// Mitsubishi GX Developer project: PLC_PCO520L2   PLC: Q06UDEH

PROGRAM OUTPUT
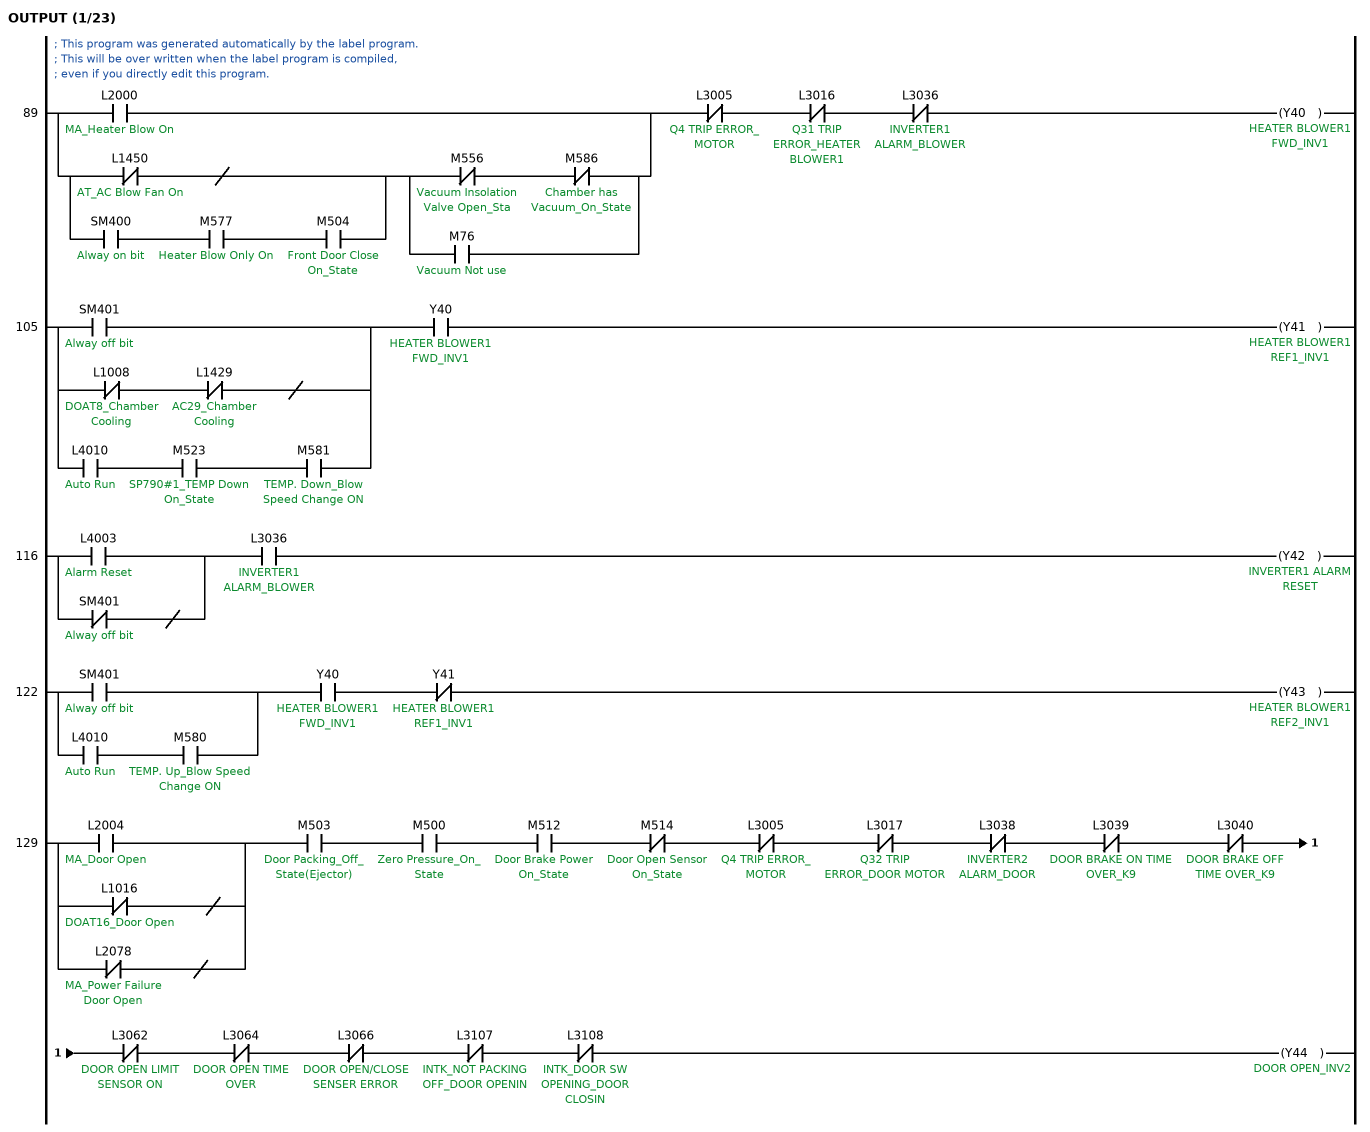
; This program was generated automatically by the label program.
; This will be over written when the label program is compiled,
; even if you directly edit this program.
89    LD      L2000  ; MA_Heater Blow On
      LDI     L1450  ; AT_AC Blow Fan On
      INV
      LD      SM400  ; Alway on bit
      AND     M577  ; Heater Blow Only On
      AND     M504  ; Front Door Close On_State
      ORB
      LDI     M556  ; Vacuum Insolation Valve Open_Sta
      ANI     M586  ; Chamber has Vacuum_On_State
      OR      M76  ; Vacuum Not use
      ANB
      ORB
      ANI     L3005  ; Q4 TRIP ERROR_MOTOR
      ANI     L3016  ; Q31 TRIP ERROR_HEATER BLOWER1
      ANI     L3036  ; INVERTER1 ALARM_BLOWER
      OUT     Y40  ; HEATER BLOWER1 FWD_INV1
105   LD      SM401  ; Alway off bit
      LDI     L1008  ; DOAT8_Chamber Cooling
      ANI     L1429  ; AC29_Chamber Cooling
      INV
      ORB
      LD      L4010  ; Auto Run
      AND     M523  ; SP790#1_TEMP Down On_State
      AND     M581  ; TEMP. Down_Blow Speed Change ON
      ORB
      AND     Y40  ; HEATER BLOWER1 FWD_INV1
      OUT     Y41  ; HEATER BLOWER1 REF1_INV1
116   LD      L4003  ; Alarm Reset
      LDI     SM401  ; Alway off bit
      INV
      ORB
      AND     L3036  ; INVERTER1 ALARM_BLOWER
      OUT     Y42  ; INVERTER1 ALARM RESET
122   LD      SM401  ; Alway off bit
      LD      L4010  ; Auto Run
      AND     M580  ; TEMP. Up_Blow Speed Change ON
      ORB
      AND     Y40  ; HEATER BLOWER1 FWD_INV1
      ANI     Y41  ; HEATER BLOWER1 REF1_INV1
      OUT     Y43  ; HEATER BLOWER1 REF2_INV1
129   LD      L2004  ; MA_Door Open
      LDI     L1016  ; DOAT16_Door Open
      INV
      ORB
      LDI     L2078  ; MA_Power Failure Door Open
      INV
      ORB
      AND     M503  ; Door Packing_Off_State(Ejector)
      AND     M500  ; Zero Pressure_On_State
      AND     M512  ; Door Brake Power On_State
      ANI     M514  ; Door Open Sensor On_State
      ANI     L3005  ; Q4 TRIP ERROR_MOTOR
      ANI     L3017  ; Q32 TRIP ERROR_DOOR MOTOR
      ANI     L3038  ; INVERTER2 ALARM_DOOR
      ANI     L3039  ; DOOR BRAKE ON TIME OVER_K9
      ANI     L3040  ; DOOR BRAKE OFF TIME OVER_K9
      ANI     L3062  ; DOOR OPEN LIMIT SENSOR ON
      ANI     L3064  ; DOOR OPEN TIME OVER
      ANI     L3066  ; DOOR OPEN/CLOSE SENSER ERROR
      ANI     L3107  ; INTK_NOT PACKING OFF_DOOR OPENIN
      ANI     L3108  ; INTK_DOOR SW OPENING_DOOR CLOSIN
      OUT     Y44  ; DOOR OPEN_INV2
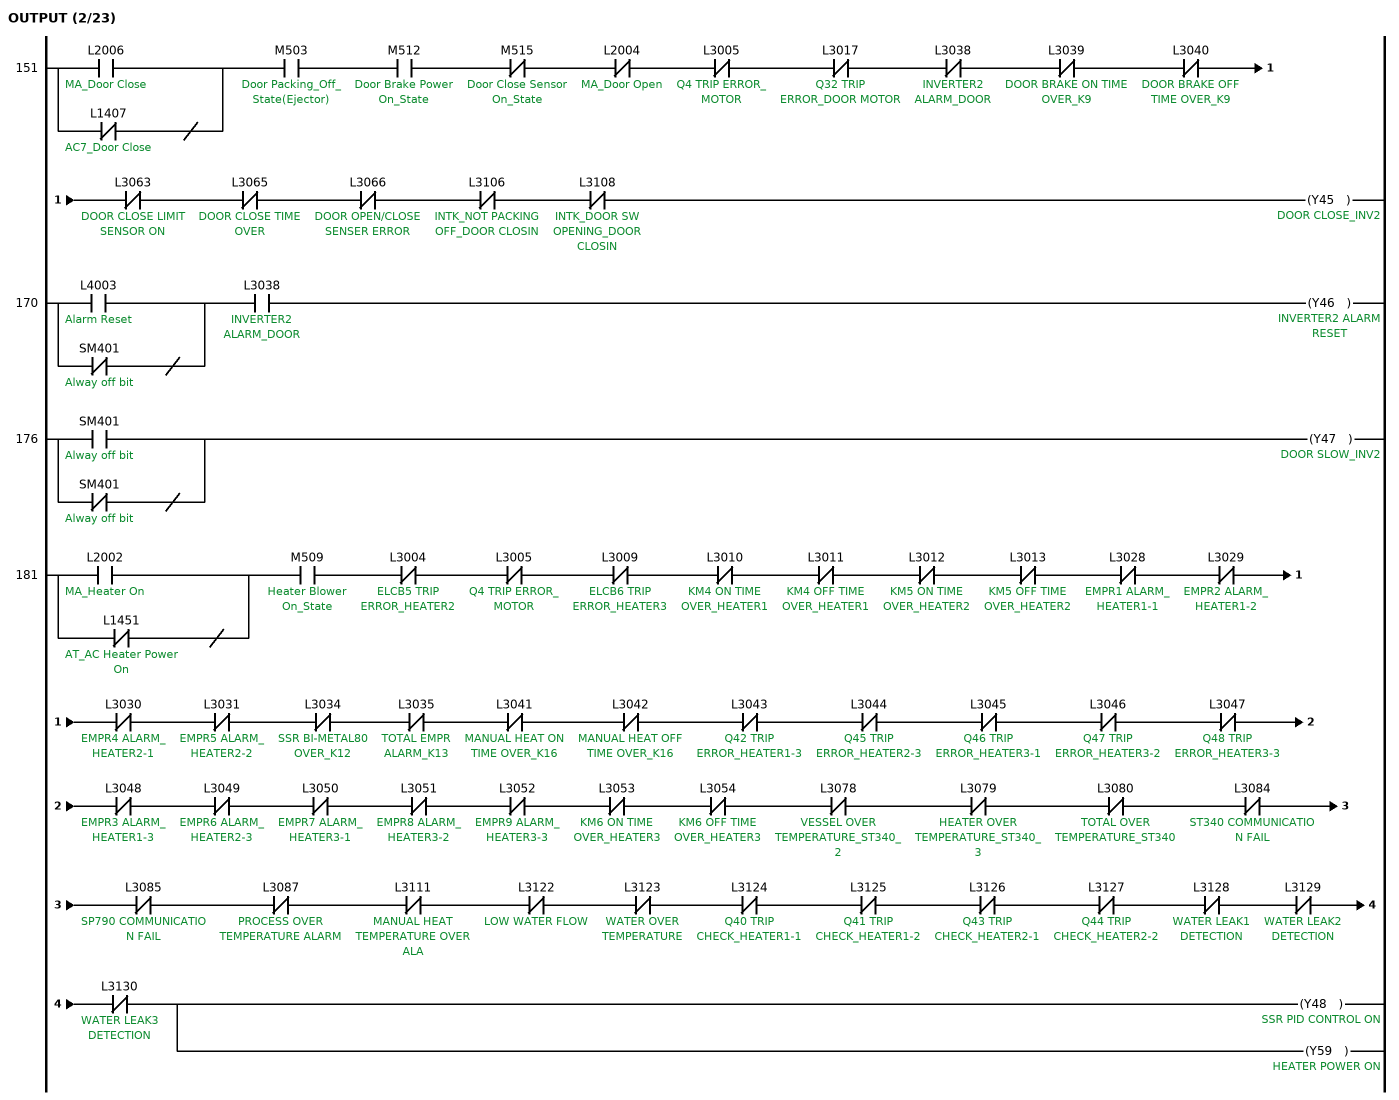
151   LD      L2006  ; MA_Door Close
      LDI     L1407  ; AC7_Door Close
      INV
      ORB
      AND     M503  ; Door Packing_Off_State(Ejector)
      AND     M512  ; Door Brake Power On_State
      ANI     M515  ; Door Close Sensor On_State
      ANI     L2004  ; MA_Door Open
      ANI     L3005  ; Q4 TRIP ERROR_MOTOR
      ANI     L3017  ; Q32 TRIP ERROR_DOOR MOTOR
      ANI     L3038  ; INVERTER2 ALARM_DOOR
      ANI     L3039  ; DOOR BRAKE ON TIME OVER_K9
      ANI     L3040  ; DOOR BRAKE OFF TIME OVER_K9
      ANI     L3063  ; DOOR CLOSE LIMIT SENSOR ON
      ANI     L3065  ; DOOR CLOSE TIME OVER
      ANI     L3066  ; DOOR OPEN/CLOSE SENSER ERROR
      ANI     L3106  ; INTK_NOT PACKING OFF_DOOR CLOSIN
      ANI     L3108  ; INTK_DOOR SW OPENING_DOOR CLOSIN
      OUT     Y45  ; DOOR CLOSE_INV2
170   LD      L4003  ; Alarm Reset
      LDI     SM401  ; Alway off bit
      INV
      ORB
      AND     L3038  ; INVERTER2 ALARM_DOOR
      OUT     Y46  ; INVERTER2 ALARM RESET
176   LD      SM401  ; Alway off bit
      LDI     SM401  ; Alway off bit
      INV
      ORB
      OUT     Y47  ; DOOR SLOW_INV2
181   LD      L2002  ; MA_Heater On
      LDI     L1451  ; AT_AC Heater Power On
      INV
      ORB
      AND     M509  ; Heater Blower On_State
      ANI     L3004  ; ELCB5 TRIP ERROR_HEATER2
      ANI     L3005  ; Q4 TRIP ERROR_MOTOR
      ANI     L3009  ; ELCB6 TRIP ERROR_HEATER3
      ANI     L3010  ; KM4 ON TIME OVER_HEATER1
      ANI     L3011  ; KM4 OFF TIME OVER_HEATER1
      ANI     L3012  ; KM5 ON TIME OVER_HEATER2
      ANI     L3013  ; KM5 OFF TIME OVER_HEATER2
      ANI     L3028  ; EMPR1 ALARM_HEATER1-1
      ANI     L3029  ; EMPR2 ALARM_HEATER1-2
      ANI     L3030  ; EMPR4 ALARM_HEATER2-1
      ANI     L3031  ; EMPR5 ALARM_HEATER2-2
      ANI     L3034  ; SSR BI-METAL80 OVER_K12
      ANI     L3035  ; TOTAL EMPR ALARM_K13
      ANI     L3041  ; MANUAL HEAT ON TIME OVER_K16
      ANI     L3042  ; MANUAL HEAT OFF TIME OVER_K16
      ANI     L3043  ; Q42 TRIP ERROR_HEATER1-3
      ANI     L3044  ; Q45 TRIP ERROR_HEATER2-3
      ANI     L3045  ; Q46 TRIP ERROR_HEATER3-1
      ANI     L3046  ; Q47 TRIP ERROR_HEATER3-2
      ANI     L3047  ; Q48 TRIP ERROR_HEATER3-3
      ANI     L3048  ; EMPR3 ALARM_HEATER1-3
      ANI     L3049  ; EMPR6 ALARM_HEATER2-3
      ANI     L3050  ; EMPR7 ALARM_HEATER3-1
      ANI     L3051  ; EMPR8 ALARM_HEATER3-2
      ANI     L3052  ; EMPR9 ALARM_HEATER3-3
      ANI     L3053  ; KM6 ON TIME OVER_HEATER3
      ANI     L3054  ; KM6 OFF TIME OVER_HEATER3
      ANI     L3078  ; VESSEL OVER TEMPERATURE_ST340_2
      ANI     L3079  ; HEATER OVER TEMPERATURE_ST340_3
      ANI     L3080  ; TOTAL OVER TEMPERATURE_ST340
      ANI     L3084  ; ST340 COMMUNICATION FAIL
      ANI     L3085  ; SP790 COMMUNICATION FAIL
      ANI     L3087  ; PROCESS OVER TEMPERATURE ALARM
      ANI     L3111  ; MANUAL HEAT TEMPERATURE OVER ALA
      ANI     L3122  ; LOW WATER FLOW
      ANI     L3123  ; WATER OVER TEMPERATURE
      ANI     L3124  ; Q40 TRIP CHECK_HEATER1-1
      ANI     L3125  ; Q41 TRIP CHECK_HEATER1-2
      ANI     L3126  ; Q43 TRIP CHECK_HEATER2-1
      ANI     L3127  ; Q44 TRIP CHECK_HEATER2-2
      ANI     L3128  ; WATER LEAK1 DETECTION
      ANI     L3129  ; WATER LEAK2 DETECTION
      ANI     L3130  ; WATER LEAK3 DETECTION
      OUT     Y48  ; SSR PID CONTROL ON
      OUT     Y59  ; HEATER POWER ON
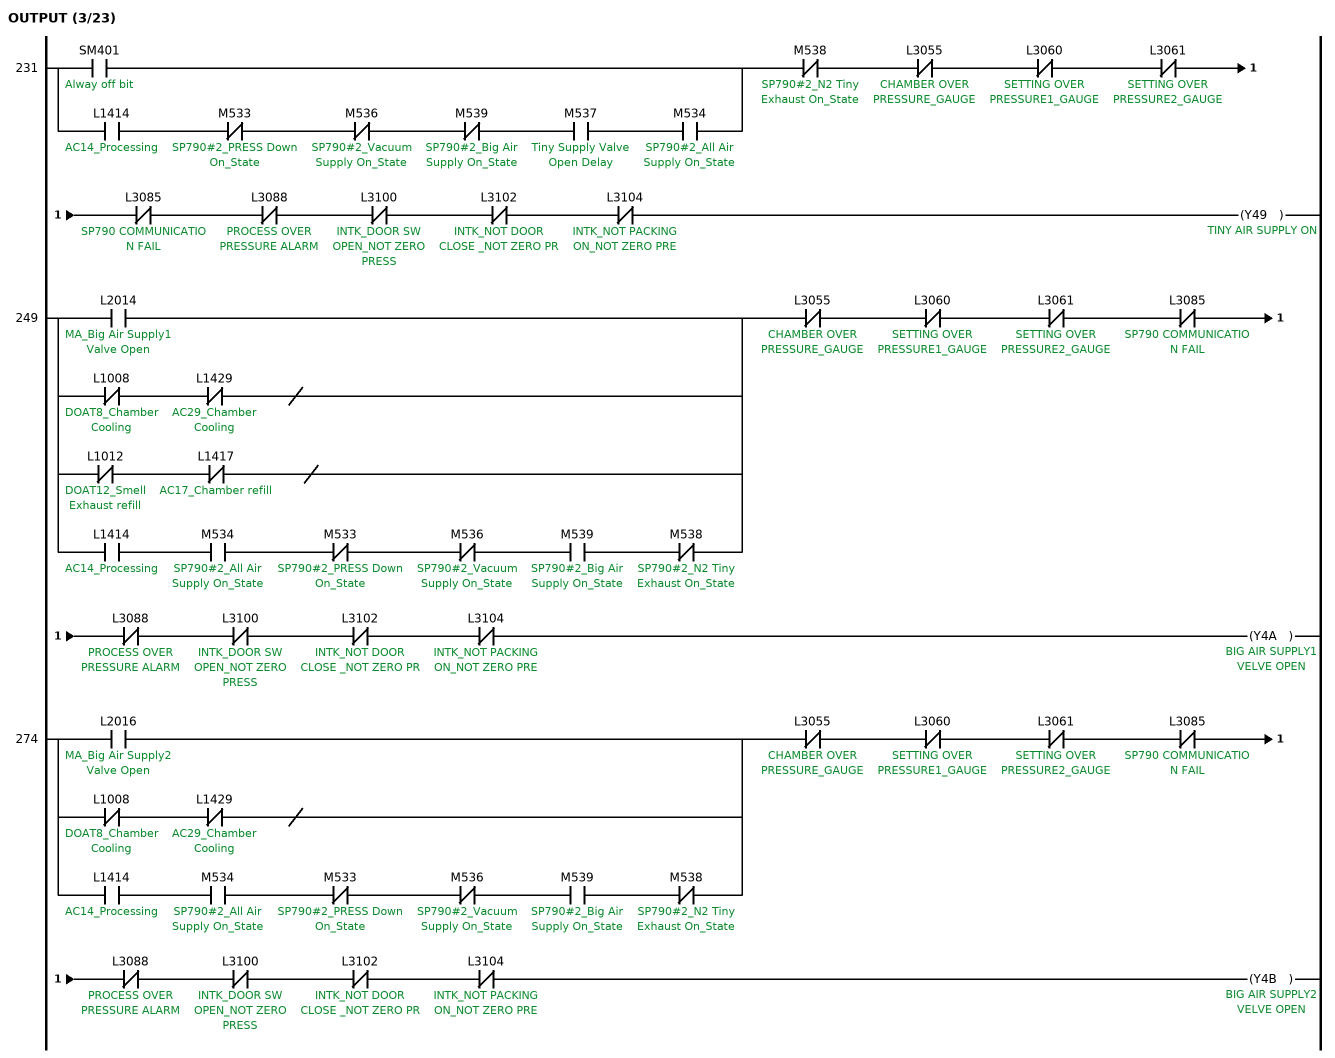
231   LD      SM401  ; Alway off bit
      LD      L1414  ; AC14_Processing
      ANI     M533  ; SP790#2_PRESS Down On_State
      ANI     M536  ; SP790#2_Vacuum Supply On_State
      ANI     M539  ; SP790#2_Big Air Supply On_State
      AND     M537  ; Tiny Supply Valve Open Delay
      AND     M534  ; SP790#2_All Air Supply On_State
      ORB
      ANI     M538  ; SP790#2_N2 Tiny Exhaust On_State
      ANI     L3055  ; CHAMBER OVER PRESSURE_GAUGE
      ANI     L3060  ; SETTING OVER PRESSURE1_GAUGE
      ANI     L3061  ; SETTING OVER PRESSURE2_GAUGE
      ANI     L3085  ; SP790 COMMUNICATION FAIL
      ANI     L3088  ; PROCESS OVER PRESSURE ALARM
      ANI     L3100  ; INTK_DOOR SW OPEN_NOT ZERO PRESS
      ANI     L3102  ; INTK_NOT DOOR CLOSE _NOT ZERO PR
      ANI     L3104  ; INTK_NOT PACKING ON_NOT ZERO PRE
      OUT     Y49  ; TINY AIR SUPPLY ON
249   LD      L2014  ; MA_Big Air Supply1 Valve Open
      LDI     L1008  ; DOAT8_Chamber Cooling
      ANI     L1429  ; AC29_Chamber Cooling
      INV
      ORB
      LDI     L1012  ; DOAT12_Smell Exhaust refill
      ANI     L1417  ; AC17_Chamber refill
      INV
      ORB
      LD      L1414  ; AC14_Processing
      AND     M534  ; SP790#2_All Air Supply On_State
      ANI     M533  ; SP790#2_PRESS Down On_State
      ANI     M536  ; SP790#2_Vacuum Supply On_State
      AND     M539  ; SP790#2_Big Air Supply On_State
      ANI     M538  ; SP790#2_N2 Tiny Exhaust On_State
      ORB
      ANI     L3055  ; CHAMBER OVER PRESSURE_GAUGE
      ANI     L3060  ; SETTING OVER PRESSURE1_GAUGE
      ANI     L3061  ; SETTING OVER PRESSURE2_GAUGE
      ANI     L3085  ; SP790 COMMUNICATION FAIL
      ANI     L3088  ; PROCESS OVER PRESSURE ALARM
      ANI     L3100  ; INTK_DOOR SW OPEN_NOT ZERO PRESS
      ANI     L3102  ; INTK_NOT DOOR CLOSE _NOT ZERO PR
      ANI     L3104  ; INTK_NOT PACKING ON_NOT ZERO PRE
      OUT     Y4A  ; BIG AIR SUPPLY1 VELVE OPEN
274   LD      L2016  ; MA_Big Air Supply2 Valve Open
      LDI     L1008  ; DOAT8_Chamber Cooling
      ANI     L1429  ; AC29_Chamber Cooling
      INV
      ORB
      LD      L1414  ; AC14_Processing
      AND     M534  ; SP790#2_All Air Supply On_State
      ANI     M533  ; SP790#2_PRESS Down On_State
      ANI     M536  ; SP790#2_Vacuum Supply On_State
      AND     M539  ; SP790#2_Big Air Supply On_State
      ANI     M538  ; SP790#2_N2 Tiny Exhaust On_State
      ORB
      ANI     L3055  ; CHAMBER OVER PRESSURE_GAUGE
      ANI     L3060  ; SETTING OVER PRESSURE1_GAUGE
      ANI     L3061  ; SETTING OVER PRESSURE2_GAUGE
      ANI     L3085  ; SP790 COMMUNICATION FAIL
      ANI     L3088  ; PROCESS OVER PRESSURE ALARM
      ANI     L3100  ; INTK_DOOR SW OPEN_NOT ZERO PRESS
      ANI     L3102  ; INTK_NOT DOOR CLOSE _NOT ZERO PR
      ANI     L3104  ; INTK_NOT PACKING ON_NOT ZERO PRE
      OUT     Y4B  ; BIG AIR SUPPLY2 VELVE OPEN
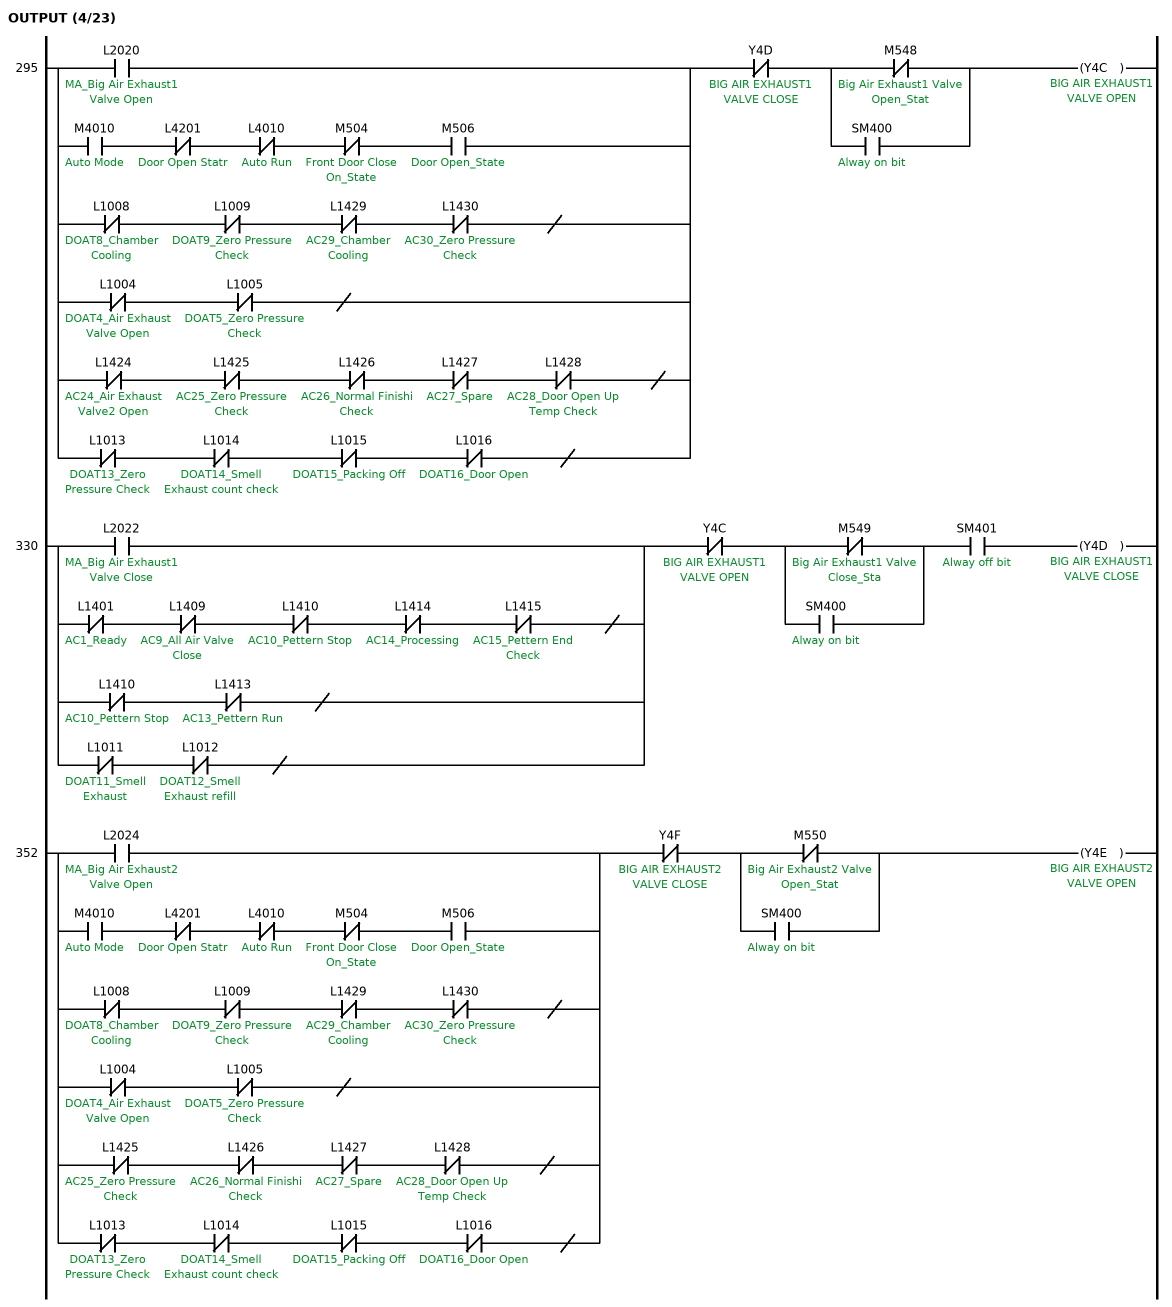
295   LD      L2020  ; MA_Big Air Exhaust1 Valve Open
      LD      M4010  ; Auto Mode
      ANI     L4201  ; Door Open Statr
      ANI     L4010  ; Auto Run
      ANI     M504  ; Front Door Close On_State
      AND     M506  ; Door Open_State
      ORB
      LDI     L1008  ; DOAT8_Chamber Cooling
      ANI     L1009  ; DOAT9_Zero Pressure Check
      ANI     L1429  ; AC29_Chamber Cooling
      ANI     L1430  ; AC30_Zero Pressure Check
      INV
      ORB
      LDI     L1004  ; DOAT4_Air Exhaust Valve Open
      ANI     L1005  ; DOAT5_Zero Pressure Check
      INV
      ORB
      LDI     L1424  ; AC24_Air Exhaust Valve2 Open
      ANI     L1425  ; AC25_Zero Pressure Check
      ANI     L1426  ; AC26_Normal Finishi Check
      ANI     L1427  ; AC27_Spare
      ANI     L1428  ; AC28_Door Open Up Temp Check
      INV
      ORB
      LDI     L1013  ; DOAT13_Zero Pressure Check
      ANI     L1014  ; DOAT14_Smell Exhaust count check
      ANI     L1015  ; DOAT15_Packing Off
      ANI     L1016  ; DOAT16_Door Open
      INV
      ORB
      ANI     Y4D  ; BIG AIR EXHAUST1 VALVE CLOSE
      LDI     M548  ; Big Air Exhaust1 Valve Open_Stat
      OR      SM400  ; Alway on bit
      ANB
      OUT     Y4C  ; BIG AIR EXHAUST1 VALVE OPEN
330   LD      L2022  ; MA_Big Air Exhaust1 Valve Close
      LDI     L1401  ; AC1_Ready
      ANI     L1409  ; AC9_All Air Valve Close
      ANI     L1410  ; AC10_Pettern Stop
      ANI     L1414  ; AC14_Processing
      ANI     L1415  ; AC15_Pettern End Check
      INV
      ORB
      LDI     L1410  ; AC10_Pettern Stop
      ANI     L1413  ; AC13_Pettern Run
      INV
      ORB
      LDI     L1011  ; DOAT11_Smell Exhaust
      ANI     L1012  ; DOAT12_Smell Exhaust refill
      INV
      ORB
      ANI     Y4C  ; BIG AIR EXHAUST1 VALVE OPEN
      LDI     M549  ; Big Air Exhaust1 Valve Close_Sta
      OR      SM400  ; Alway on bit
      ANB
      AND     SM401  ; Alway off bit
      OUT     Y4D  ; BIG AIR EXHAUST1 VALVE CLOSE
352   LD      L2024  ; MA_Big Air Exhaust2 Valve Open
      LD      M4010  ; Auto Mode
      ANI     L4201  ; Door Open Statr
      ANI     L4010  ; Auto Run
      ANI     M504  ; Front Door Close On_State
      AND     M506  ; Door Open_State
      ORB
      LDI     L1008  ; DOAT8_Chamber Cooling
      ANI     L1009  ; DOAT9_Zero Pressure Check
      ANI     L1429  ; AC29_Chamber Cooling
      ANI     L1430  ; AC30_Zero Pressure Check
      INV
      ORB
      LDI     L1004  ; DOAT4_Air Exhaust Valve Open
      ANI     L1005  ; DOAT5_Zero Pressure Check
      INV
      ORB
      LDI     L1425  ; AC25_Zero Pressure Check
      ANI     L1426  ; AC26_Normal Finishi Check
      ANI     L1427  ; AC27_Spare
      ANI     L1428  ; AC28_Door Open Up Temp Check
      INV
      ORB
      LDI     L1013  ; DOAT13_Zero Pressure Check
      ANI     L1014  ; DOAT14_Smell Exhaust count check
      ANI     L1015  ; DOAT15_Packing Off
      ANI     L1016  ; DOAT16_Door Open
      INV
      ORB
      ANI     Y4F  ; BIG AIR EXHAUST2 VALVE CLOSE
      LDI     M550  ; Big Air Exhaust2 Valve Open_Stat
      OR      SM400  ; Alway on bit
      ANB
      OUT     Y4E  ; BIG AIR EXHAUST2 VALVE OPEN
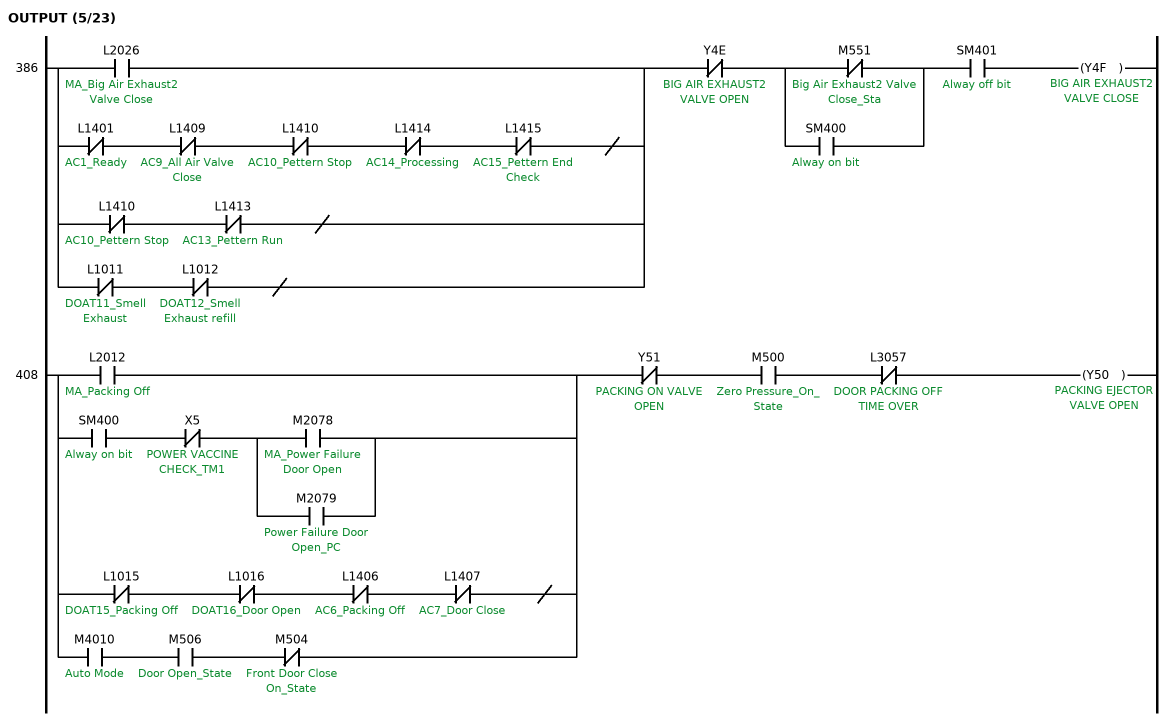
386   LD      L2026  ; MA_Big Air Exhaust2 Valve Close
      LDI     L1401  ; AC1_Ready
      ANI     L1409  ; AC9_All Air Valve Close
      ANI     L1410  ; AC10_Pettern Stop
      ANI     L1414  ; AC14_Processing
      ANI     L1415  ; AC15_Pettern End Check
      INV
      ORB
      LDI     L1410  ; AC10_Pettern Stop
      ANI     L1413  ; AC13_Pettern Run
      INV
      ORB
      LDI     L1011  ; DOAT11_Smell Exhaust
      ANI     L1012  ; DOAT12_Smell Exhaust refill
      INV
      ORB
      ANI     Y4E  ; BIG AIR EXHAUST2 VALVE OPEN
      LDI     M551  ; Big Air Exhaust2 Valve Close_Sta
      OR      SM400  ; Alway on bit
      ANB
      AND     SM401  ; Alway off bit
      OUT     Y4F  ; BIG AIR EXHAUST2 VALVE CLOSE
408   LD      L2012  ; MA_Packing Off
      LD      SM400  ; Alway on bit
      ANI     X5  ; POWER VACCINE CHECK_TM1
      LD      M2078  ; MA_Power Failure Door Open
      OR      M2079  ; Power Failure Door Open_PC
      ANB
      ORB
      LDI     L1015  ; DOAT15_Packing Off
      ANI     L1016  ; DOAT16_Door Open
      ANI     L1406  ; AC6_Packing Off
      ANI     L1407  ; AC7_Door Close
      INV
      ORB
      LD      M4010  ; Auto Mode
      AND     M506  ; Door Open_State
      ANI     M504  ; Front Door Close On_State
      ORB
      ANI     Y51  ; PACKING ON VALVE OPEN
      AND     M500  ; Zero Pressure_On_State
      ANI     L3057  ; DOOR PACKING OFF TIME OVER
      OUT     Y50  ; PACKING EJECTOR VALVE OPEN
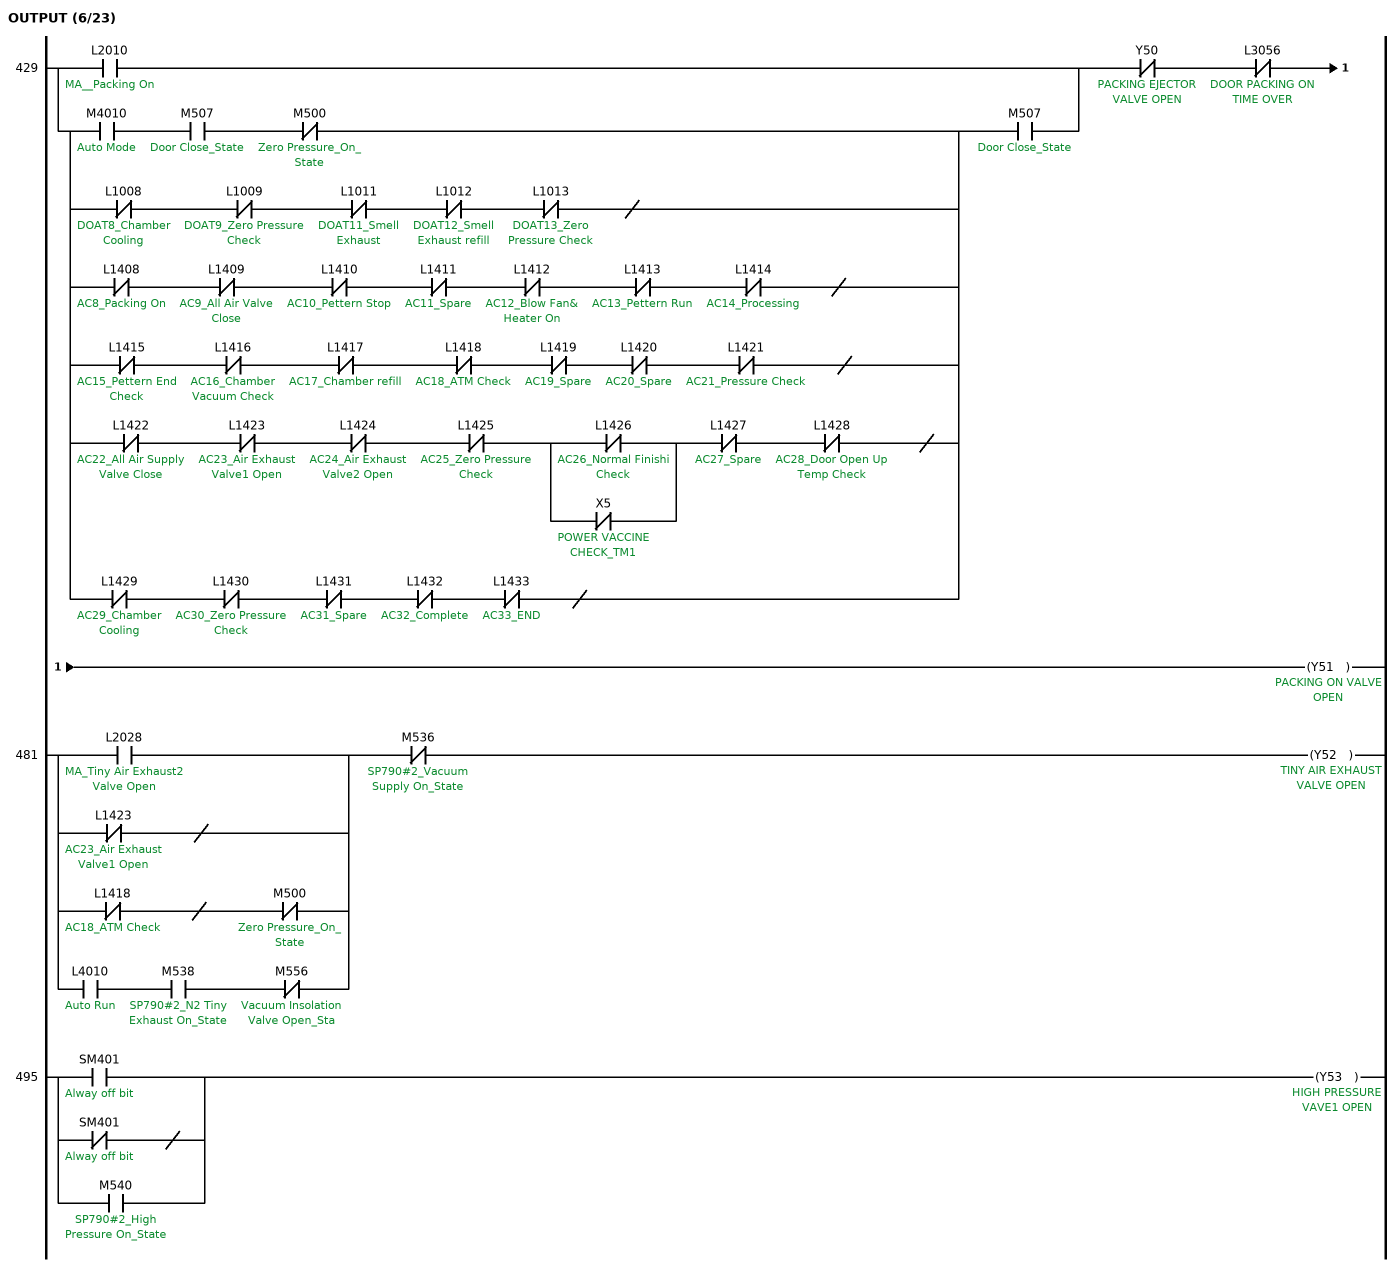
429   LD      L2010  ; MA__Packing On
      LD      M4010  ; Auto Mode
      AND     M507  ; Door Close_State
      ANI     M500  ; Zero Pressure_On_State
      LDI     L1008  ; DOAT8_Chamber Cooling
      ANI     L1009  ; DOAT9_Zero Pressure Check
      ANI     L1011  ; DOAT11_Smell Exhaust
      ANI     L1012  ; DOAT12_Smell Exhaust refill
      ANI     L1013  ; DOAT13_Zero Pressure Check
      INV
      ORB
      LDI     L1408  ; AC8_Packing On
      ANI     L1409  ; AC9_All Air Valve Close
      ANI     L1410  ; AC10_Pettern Stop
      ANI     L1411  ; AC11_Spare
      ANI     L1412  ; AC12_Blow Fan& Heater On
      ANI     L1413  ; AC13_Pettern Run
      ANI     L1414  ; AC14_Processing
      INV
      ORB
      LDI     L1415  ; AC15_Pettern End Check
      ANI     L1416  ; AC16_Chamber Vacuum Check
      ANI     L1417  ; AC17_Chamber refill
      ANI     L1418  ; AC18_ATM Check
      ANI     L1419  ; AC19_Spare
      ANI     L1420  ; AC20_Spare
      ANI     L1421  ; AC21_Pressure Check
      INV
      ORB
      LDI     L1422  ; AC22_All Air Supply Valve Close
      ANI     L1423  ; AC23_Air Exhaust Valve1 Open
      ANI     L1424  ; AC24_Air Exhaust Valve2 Open
      ANI     L1425  ; AC25_Zero Pressure Check
      LDI     L1426  ; AC26_Normal Finishi Check
      ORI     X5  ; POWER VACCINE CHECK_TM1
      ANB
      ANI     L1427  ; AC27_Spare
      ANI     L1428  ; AC28_Door Open Up Temp Check
      INV
      ORB
      LDI     L1429  ; AC29_Chamber Cooling
      ANI     L1430  ; AC30_Zero Pressure Check
      ANI     L1431  ; AC31_Spare
      ANI     L1432  ; AC32_Complete
      ANI     L1433  ; AC33_END
      INV
      ORB
      AND     M507  ; Door Close_State
      ORB
      ANI     Y50  ; PACKING EJECTOR VALVE OPEN
      ANI     L3056  ; DOOR PACKING ON TIME OVER
      OUT     Y51  ; PACKING ON VALVE OPEN
481   LD      L2028  ; MA_Tiny Air Exhaust2 Valve Open
      LDI     L1423  ; AC23_Air Exhaust Valve1 Open
      INV
      ORB
      LDI     L1418  ; AC18_ATM Check
      INV
      ANI     M500  ; Zero Pressure_On_State
      ORB
      LD      L4010  ; Auto Run
      AND     M538  ; SP790#2_N2 Tiny Exhaust On_State
      ANI     M556  ; Vacuum Insolation Valve Open_Sta
      ORB
      ANI     M536  ; SP790#2_Vacuum Supply On_State
      OUT     Y52  ; TINY AIR EXHAUST VALVE OPEN
495   LD      SM401  ; Alway off bit
      LDI     SM401  ; Alway off bit
      INV
      ORB
      OR      M540  ; SP790#2_High Pressure On_State
      OUT     Y53  ; HIGH PRESSURE VAVE1 OPEN
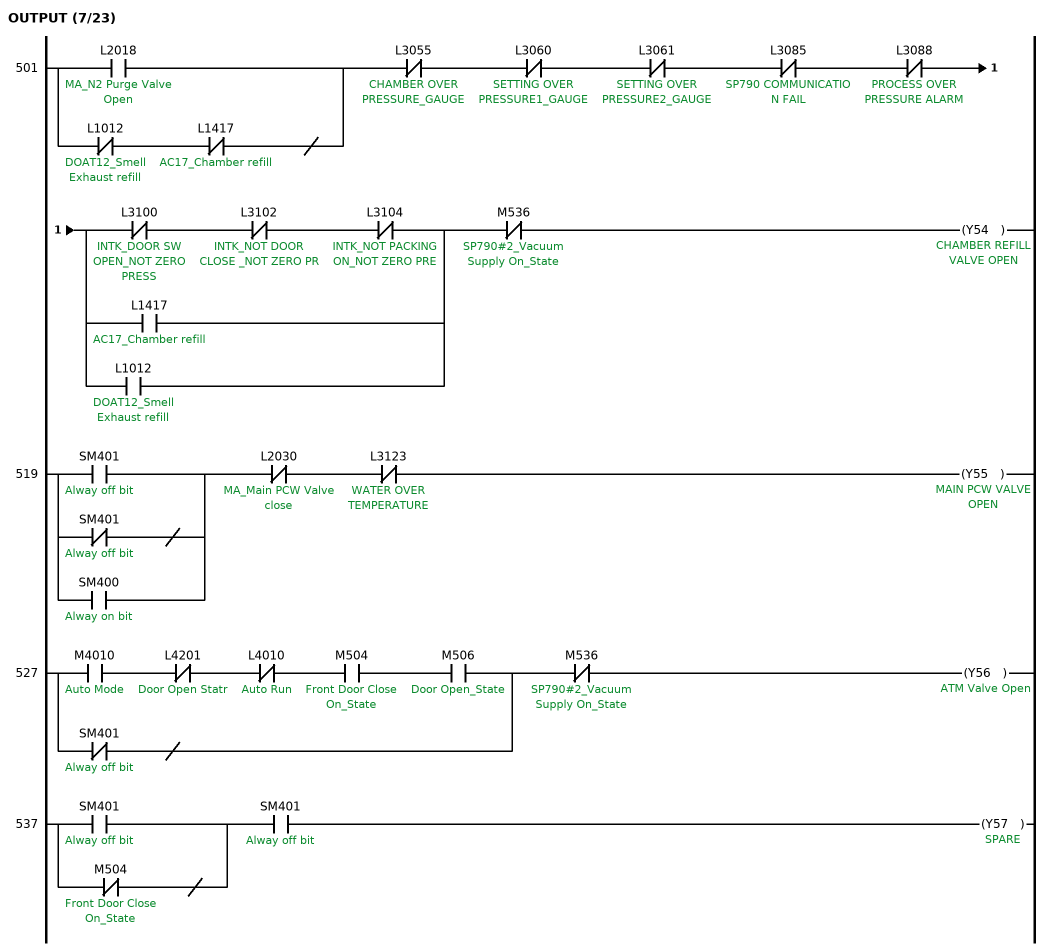
501   LD      L2018  ; MA_N2 Purge Valve Open
      LDI     L1012  ; DOAT12_Smell Exhaust refill
      ANI     L1417  ; AC17_Chamber refill
      INV
      ORB
      ANI     L3055  ; CHAMBER OVER PRESSURE_GAUGE
      ANI     L3060  ; SETTING OVER PRESSURE1_GAUGE
      ANI     L3061  ; SETTING OVER PRESSURE2_GAUGE
      ANI     L3085  ; SP790 COMMUNICATION FAIL
      ANI     L3088  ; PROCESS OVER PRESSURE ALARM
      LDI     L3100  ; INTK_DOOR SW OPEN_NOT ZERO PRESS
      ANI     L3102  ; INTK_NOT DOOR CLOSE _NOT ZERO PR
      ANI     L3104  ; INTK_NOT PACKING ON_NOT ZERO PRE
      OR      L1417  ; AC17_Chamber refill
      OR      L1012  ; DOAT12_Smell Exhaust refill
      ANB
      ANI     M536  ; SP790#2_Vacuum Supply On_State
      OUT     Y54  ; CHAMBER REFILL VALVE OPEN
519   LD      SM401  ; Alway off bit
      LDI     SM401  ; Alway off bit
      INV
      ORB
      OR      SM400  ; Alway on bit
      ANI     L2030  ; MA_Main PCW Valve close
      ANI     L3123  ; WATER OVER TEMPERATURE
      OUT     Y55  ; MAIN PCW VALVE OPEN
527   LD      M4010  ; Auto Mode
      ANI     L4201  ; Door Open Statr
      ANI     L4010  ; Auto Run
      AND     M504  ; Front Door Close On_State
      AND     M506  ; Door Open_State
      LDI     SM401  ; Alway off bit
      INV
      ORB
      ANI     M536  ; SP790#2_Vacuum Supply On_State
      OUT     Y56  ; ATM Valve Open
537   LD      SM401  ; Alway off bit
      LDI     M504  ; Front Door Close On_State
      INV
      ORB
      AND     SM401  ; Alway off bit
      OUT     Y57  ; SPARE
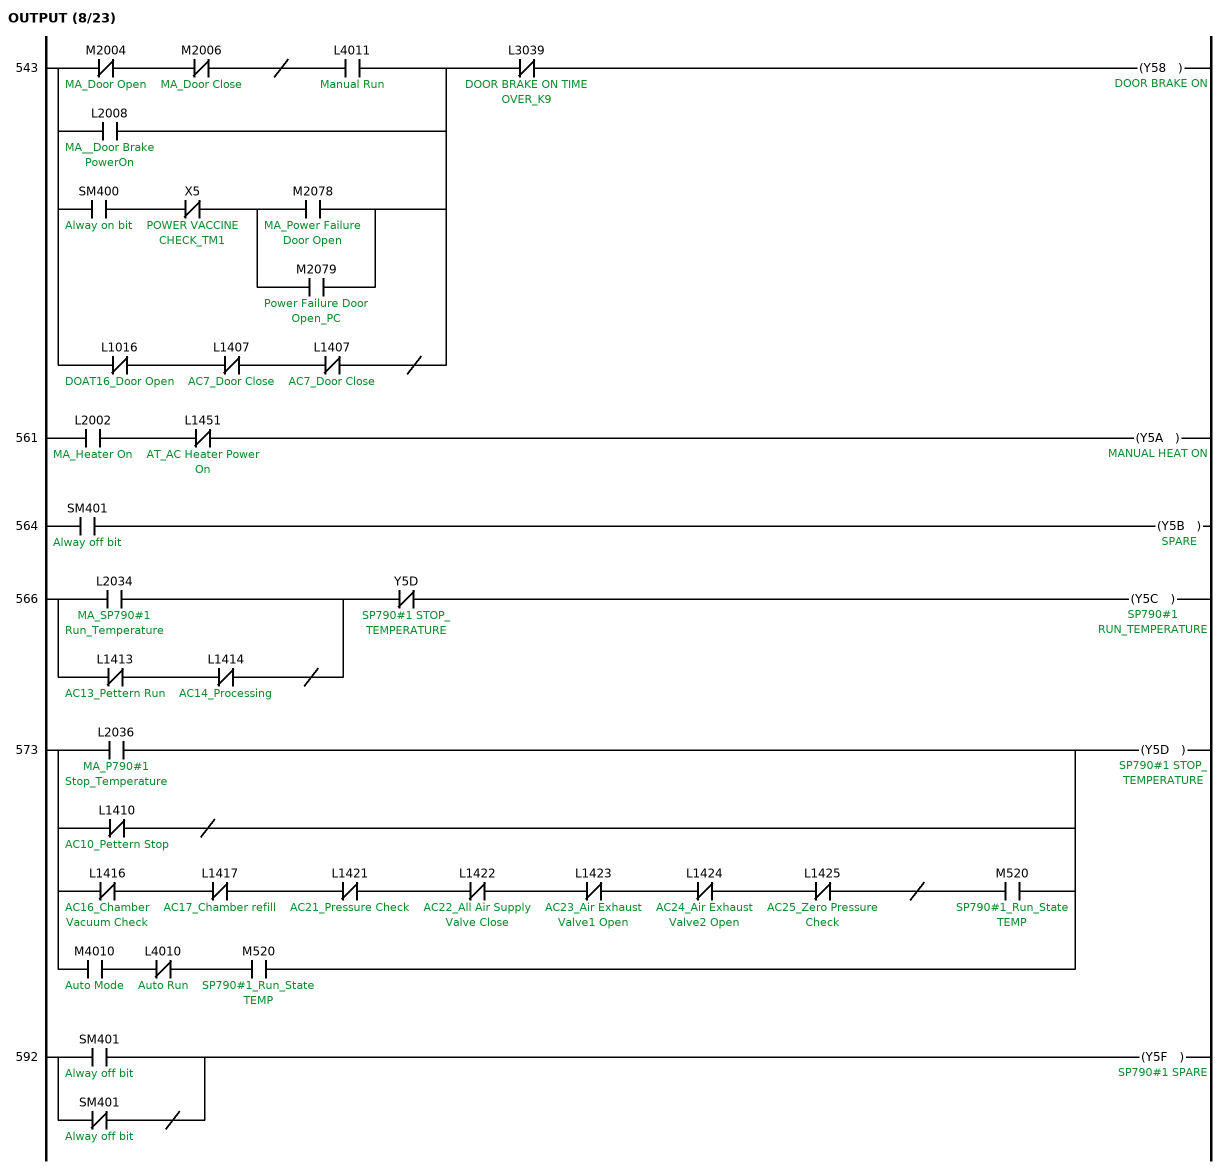
543   LDI     M2004  ; MA_Door Open
      ANI     M2006  ; MA_Door Close
      INV
      AND     L4011  ; Manual Run
      OR      L2008  ; MA__Door Brake PowerOn
      LD      SM400  ; Alway on bit
      ANI     X5  ; POWER VACCINE CHECK_TM1
      LD      M2078  ; MA_Power Failure Door Open
      OR      M2079  ; Power Failure Door Open_PC
      ANB
      ORB
      LDI     L1016  ; DOAT16_Door Open
      ANI     L1407  ; AC7_Door Close
      ANI     L1407  ; AC7_Door Close
      INV
      ORB
      ANI     L3039  ; DOOR BRAKE ON TIME OVER_K9
      OUT     Y58  ; DOOR BRAKE ON
561   LD      L2002  ; MA_Heater On
      ANI     L1451  ; AT_AC Heater Power On
      OUT     Y5A  ; MANUAL HEAT ON
564   LD      SM401  ; Alway off bit
      OUT     Y5B  ; SPARE
566   LD      L2034  ; MA_SP790#1 Run_Temperature
      LDI     L1413  ; AC13_Pettern Run
      ANI     L1414  ; AC14_Processing
      INV
      ORB
      ANI     Y5D  ; SP790#1 STOP_TEMPERATURE
      OUT     Y5C  ; SP790#1 RUN_TEMPERATURE
573   LD      L2036  ; MA_P790#1 Stop_Temperature
      LDI     L1410  ; AC10_Pettern Stop
      INV
      ORB
      LDI     L1416  ; AC16_Chamber Vacuum Check
      ANI     L1417  ; AC17_Chamber refill
      ANI     L1421  ; AC21_Pressure Check
      ANI     L1422  ; AC22_All Air Supply Valve Close
      ANI     L1423  ; AC23_Air Exhaust Valve1 Open
      ANI     L1424  ; AC24_Air Exhaust Valve2 Open
      ANI     L1425  ; AC25_Zero Pressure Check
      INV
      AND     M520  ; SP790#1_Run_State TEMP
      ORB
      LD      M4010  ; Auto Mode
      ANI     L4010  ; Auto Run
      AND     M520  ; SP790#1_Run_State TEMP
      ORB
      OUT     Y5D  ; SP790#1 STOP_TEMPERATURE
592   LD      SM401  ; Alway off bit
      LDI     SM401  ; Alway off bit
      INV
      ORB
      OUT     Y5F  ; SP790#1 SPARE
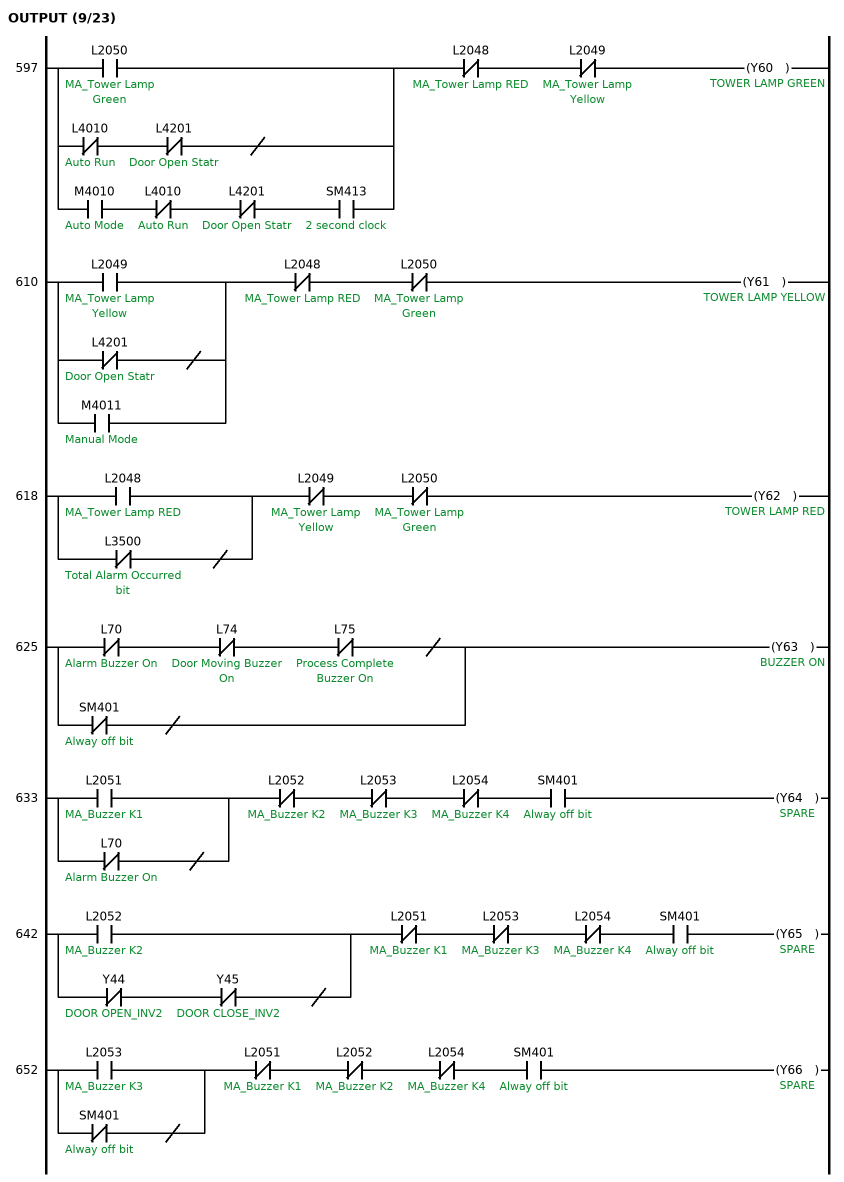
597   LD      L2050  ; MA_Tower Lamp Green
      LDI     L4010  ; Auto Run
      ANI     L4201  ; Door Open Statr
      INV
      ORB
      LD      M4010  ; Auto Mode
      ANI     L4010  ; Auto Run
      ANI     L4201  ; Door Open Statr
      AND     SM413  ; 2 second clock
      ORB
      ANI     L2048  ; MA_Tower Lamp RED
      ANI     L2049  ; MA_Tower Lamp Yellow
      OUT     Y60  ; TOWER LAMP GREEN
610   LD      L2049  ; MA_Tower Lamp Yellow
      LDI     L4201  ; Door Open Statr
      INV
      ORB
      OR      M4011  ; Manual Mode
      ANI     L2048  ; MA_Tower Lamp RED
      ANI     L2050  ; MA_Tower Lamp Green
      OUT     Y61  ; TOWER LAMP YELLOW
618   LD      L2048  ; MA_Tower Lamp RED
      LDI     L3500  ; Total Alarm Occurred bit
      INV
      ORB
      ANI     L2049  ; MA_Tower Lamp Yellow
      ANI     L2050  ; MA_Tower Lamp Green
      OUT     Y62  ; TOWER LAMP RED
625   LDI     L70  ; Alarm Buzzer On
      ANI     L74  ; Door Moving Buzzer On
      ANI     L75  ; Process Complete Buzzer On
      INV
      LDI     SM401  ; Alway off bit
      INV
      ORB
      OUT     Y63  ; BUZZER ON
633   LD      L2051  ; MA_Buzzer K1
      LDI     L70  ; Alarm Buzzer On
      INV
      ORB
      ANI     L2052  ; MA_Buzzer K2
      ANI     L2053  ; MA_Buzzer K3
      ANI     L2054  ; MA_Buzzer K4
      AND     SM401  ; Alway off bit
      OUT     Y64  ; SPARE
642   LD      L2052  ; MA_Buzzer K2
      LDI     Y44  ; DOOR OPEN_INV2
      ANI     Y45  ; DOOR CLOSE_INV2
      INV
      ORB
      ANI     L2051  ; MA_Buzzer K1
      ANI     L2053  ; MA_Buzzer K3
      ANI     L2054  ; MA_Buzzer K4
      AND     SM401  ; Alway off bit
      OUT     Y65  ; SPARE
652   LD      L2053  ; MA_Buzzer K3
      LDI     SM401  ; Alway off bit
      INV
      ORB
      ANI     L2051  ; MA_Buzzer K1
      ANI     L2052  ; MA_Buzzer K2
      ANI     L2054  ; MA_Buzzer K4
      AND     SM401  ; Alway off bit
      OUT     Y66  ; SPARE
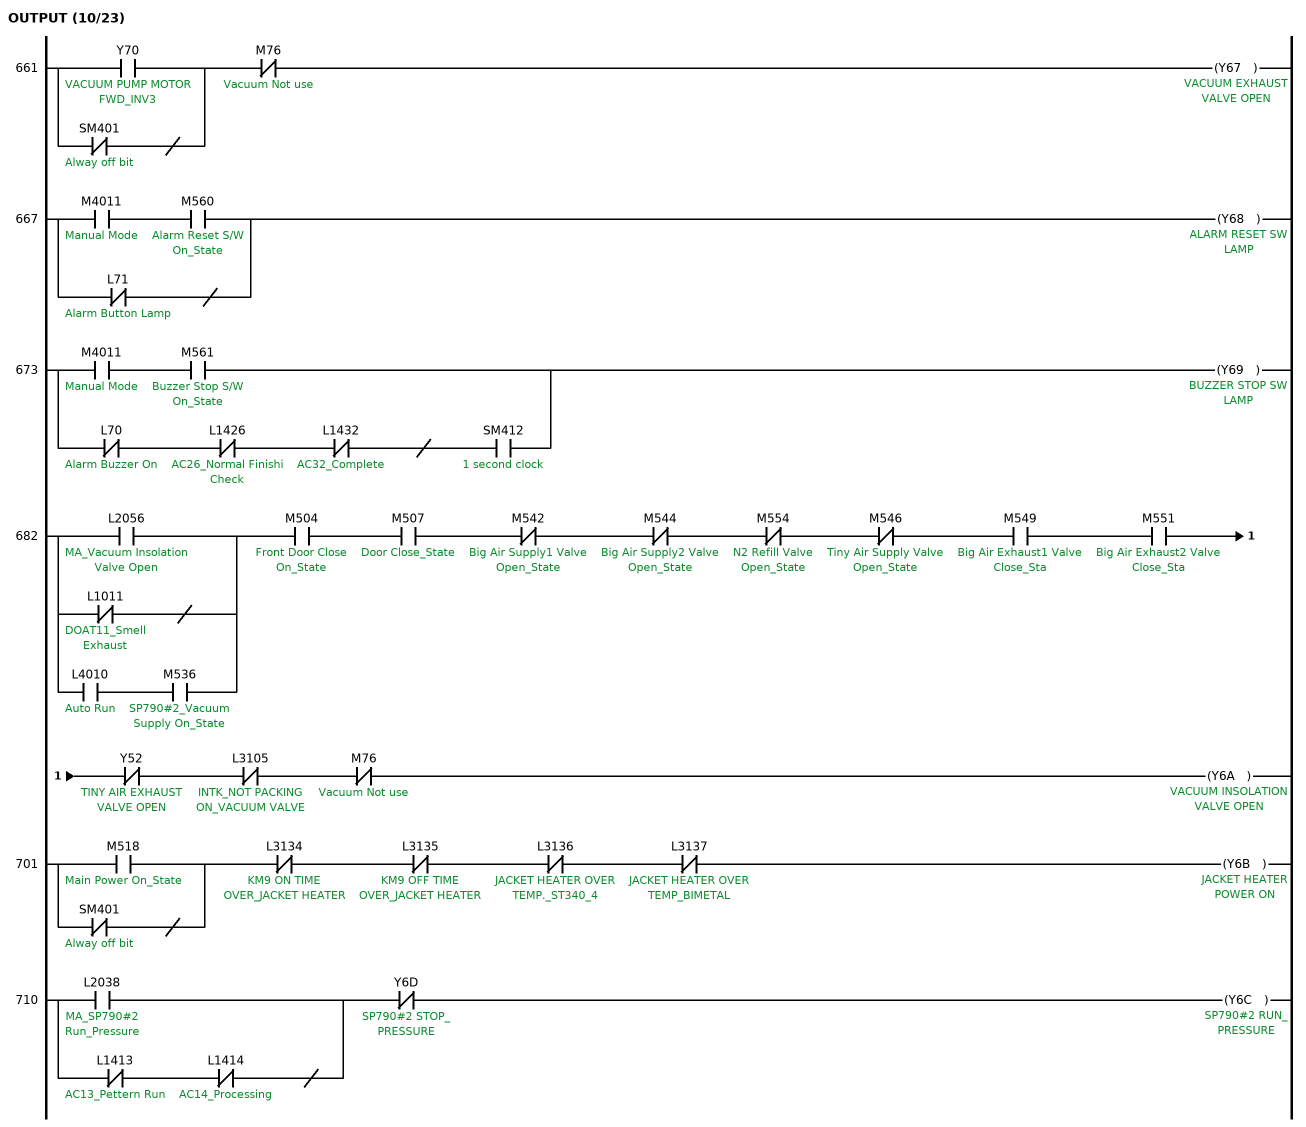
661   LD      Y70  ; VACUUM PUMP MOTOR FWD_INV3
      LDI     SM401  ; Alway off bit
      INV
      ORB
      ANI     M76  ; Vacuum Not use
      OUT     Y67  ; VACUUM EXHAUST VALVE OPEN
667   LD      M4011  ; Manual Mode
      AND     M560  ; Alarm Reset S/W On_State
      LDI     L71  ; Alarm Button Lamp
      INV
      ORB
      OUT     Y68  ; ALARM RESET SW LAMP
673   LD      M4011  ; Manual Mode
      AND     M561  ; Buzzer Stop S/W On_State
      LDI     L70  ; Alarm Buzzer On
      ANI     L1426  ; AC26_Normal Finishi Check
      ANI     L1432  ; AC32_Complete
      INV
      AND     SM412  ; 1 second clock
      ORB
      OUT     Y69  ; BUZZER STOP SW LAMP
682   LD      L2056  ; MA_Vacuum Insolation Valve Open
      LDI     L1011  ; DOAT11_Smell Exhaust
      INV
      ORB
      LD      L4010  ; Auto Run
      AND     M536  ; SP790#2_Vacuum Supply On_State
      ORB
      AND     M504  ; Front Door Close On_State
      AND     M507  ; Door Close_State
      ANI     M542  ; Big Air Supply1 Valve Open_State
      ANI     M544  ; Big Air Supply2 Valve Open_State
      ANI     M554  ; N2 Refill Valve Open_State
      ANI     M546  ; Tiny Air Supply Valve Open_State
      AND     M549  ; Big Air Exhaust1 Valve Close_Sta
      AND     M551  ; Big Air Exhaust2 Valve Close_Sta
      ANI     Y52  ; TINY AIR EXHAUST VALVE OPEN
      ANI     L3105  ; INTK_NOT PACKING ON_VACUUM VALVE
      ANI     M76  ; Vacuum Not use
      OUT     Y6A  ; VACUUM INSOLATION VALVE OPEN
701   LD      M518  ; Main Power On_State
      LDI     SM401  ; Alway off bit
      INV
      ORB
      ANI     L3134  ; KM9 ON TIME OVER_JACKET HEATER
      ANI     L3135  ; KM9 OFF TIME OVER_JACKET HEATER
      ANI     L3136  ; JACKET HEATER OVER TEMP._ST340_4
      ANI     L3137  ; JACKET HEATER OVER TEMP_BIMETAL
      OUT     Y6B  ; JACKET HEATER POWER ON
710   LD      L2038  ; MA_SP790#2 Run_Pressure
      LDI     L1413  ; AC13_Pettern Run
      ANI     L1414  ; AC14_Processing
      INV
      ORB
      ANI     Y6D  ; SP790#2 STOP_PRESSURE
      OUT     Y6C  ; SP790#2 RUN_PRESSURE
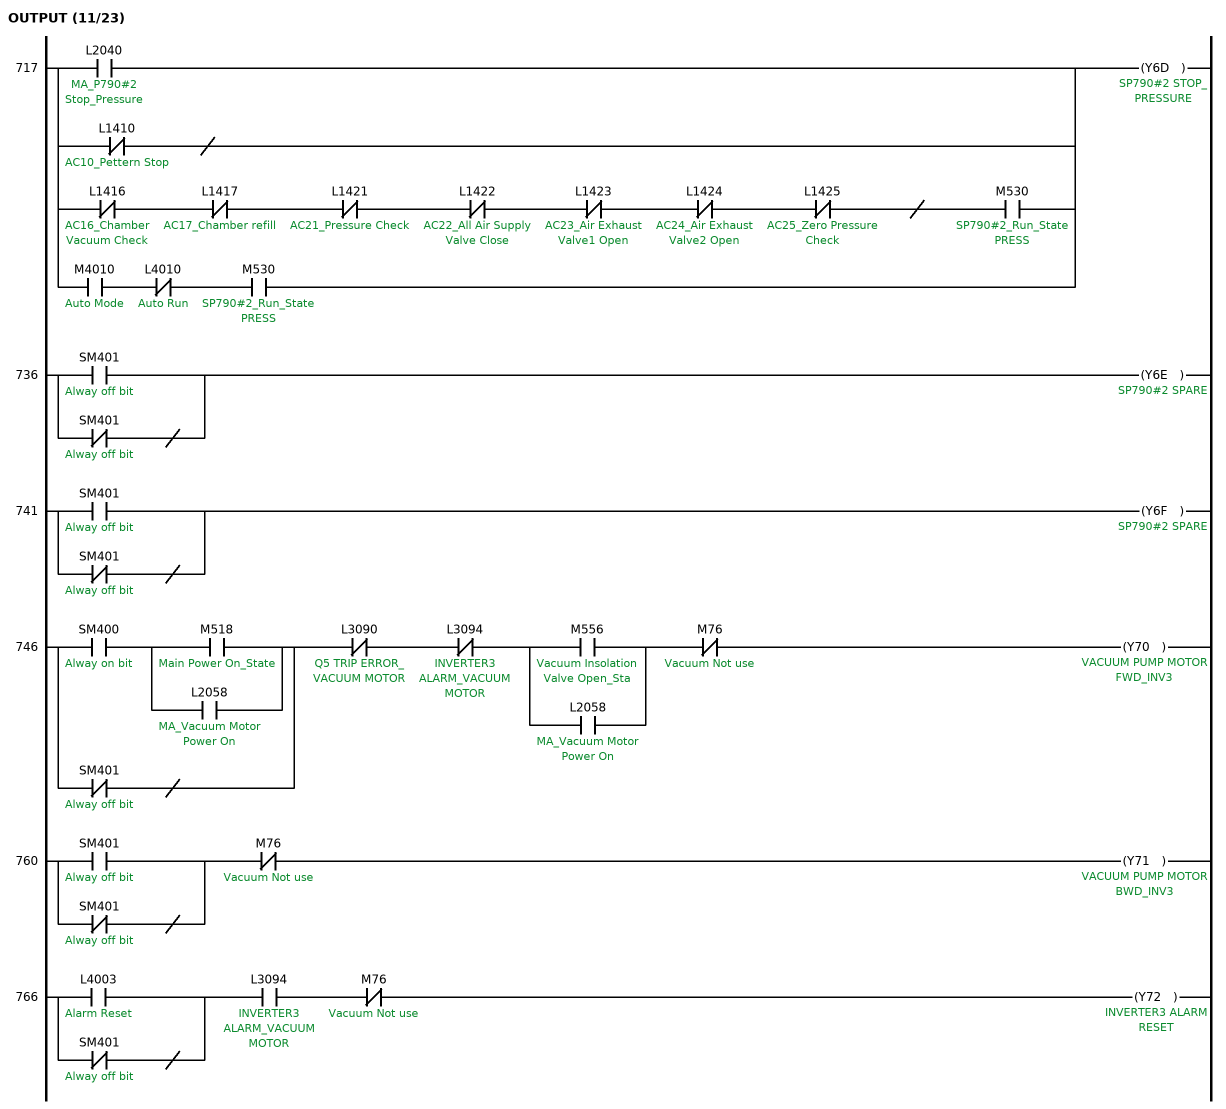
717   LD      L2040  ; MA_P790#2 Stop_Pressure
      LDI     L1410  ; AC10_Pettern Stop
      INV
      ORB
      LDI     L1416  ; AC16_Chamber Vacuum Check
      ANI     L1417  ; AC17_Chamber refill
      ANI     L1421  ; AC21_Pressure Check
      ANI     L1422  ; AC22_All Air Supply Valve Close
      ANI     L1423  ; AC23_Air Exhaust Valve1 Open
      ANI     L1424  ; AC24_Air Exhaust Valve2 Open
      ANI     L1425  ; AC25_Zero Pressure Check
      INV
      AND     M530  ; SP790#2_Run_State PRESS
      ORB
      LD      M4010  ; Auto Mode
      ANI     L4010  ; Auto Run
      AND     M530  ; SP790#2_Run_State PRESS
      ORB
      OUT     Y6D  ; SP790#2 STOP_PRESSURE
736   LD      SM401  ; Alway off bit
      LDI     SM401  ; Alway off bit
      INV
      ORB
      OUT     Y6E  ; SP790#2 SPARE
741   LD      SM401  ; Alway off bit
      LDI     SM401  ; Alway off bit
      INV
      ORB
      OUT     Y6F  ; SP790#2 SPARE
746   LD      SM400  ; Alway on bit
      LD      M518  ; Main Power On_State
      OR      L2058  ; MA_Vacuum Motor Power On
      ANB
      LDI     SM401  ; Alway off bit
      INV
      ORB
      ANI     L3090  ; Q5 TRIP ERROR_VACUUM MOTOR
      ANI     L3094  ; INVERTER3 ALARM_VACUUM MOTOR
      LD      M556  ; Vacuum Insolation Valve Open_Sta
      OR      L2058  ; MA_Vacuum Motor Power On
      ANB
      ANI     M76  ; Vacuum Not use
      OUT     Y70  ; VACUUM PUMP MOTOR FWD_INV3
760   LD      SM401  ; Alway off bit
      LDI     SM401  ; Alway off bit
      INV
      ORB
      ANI     M76  ; Vacuum Not use
      OUT     Y71  ; VACUUM PUMP MOTOR BWD_INV3
766   LD      L4003  ; Alarm Reset
      LDI     SM401  ; Alway off bit
      INV
      ORB
      AND     L3094  ; INVERTER3 ALARM_VACUUM MOTOR
      ANI     M76  ; Vacuum Not use
      OUT     Y72  ; INVERTER3 ALARM RESET
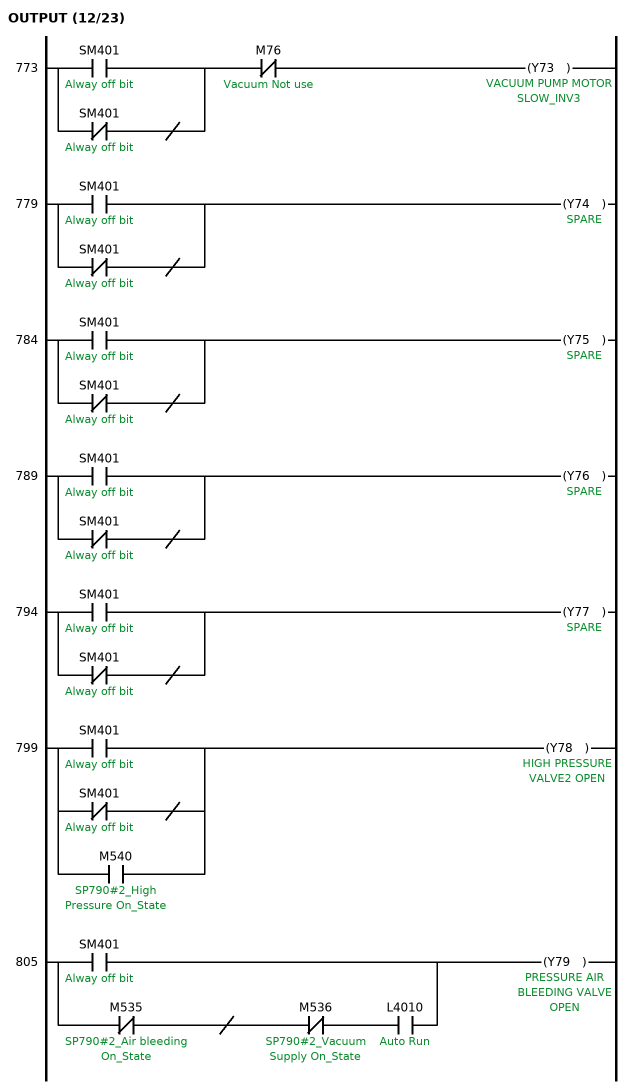
773   LD      SM401  ; Alway off bit
      LDI     SM401  ; Alway off bit
      INV
      ORB
      ANI     M76  ; Vacuum Not use
      OUT     Y73  ; VACUUM PUMP MOTOR SLOW_INV3
779   LD      SM401  ; Alway off bit
      LDI     SM401  ; Alway off bit
      INV
      ORB
      OUT     Y74  ; SPARE
784   LD      SM401  ; Alway off bit
      LDI     SM401  ; Alway off bit
      INV
      ORB
      OUT     Y75  ; SPARE
789   LD      SM401  ; Alway off bit
      LDI     SM401  ; Alway off bit
      INV
      ORB
      OUT     Y76  ; SPARE
794   LD      SM401  ; Alway off bit
      LDI     SM401  ; Alway off bit
      INV
      ORB
      OUT     Y77  ; SPARE
799   LD      SM401  ; Alway off bit
      LDI     SM401  ; Alway off bit
      INV
      ORB
      OR      M540  ; SP790#2_High Pressure On_State
      OUT     Y78  ; HIGH PRESSURE VALVE2 OPEN
805   LD      SM401  ; Alway off bit
      LDI     M535  ; SP790#2_Air bleeding On_State
      INV
      ANI     M536  ; SP790#2_Vacuum Supply On_State
      AND     L4010  ; Auto Run
      ORB
      OUT     Y79  ; PRESSURE AIR BLEEDING VALVE OPEN
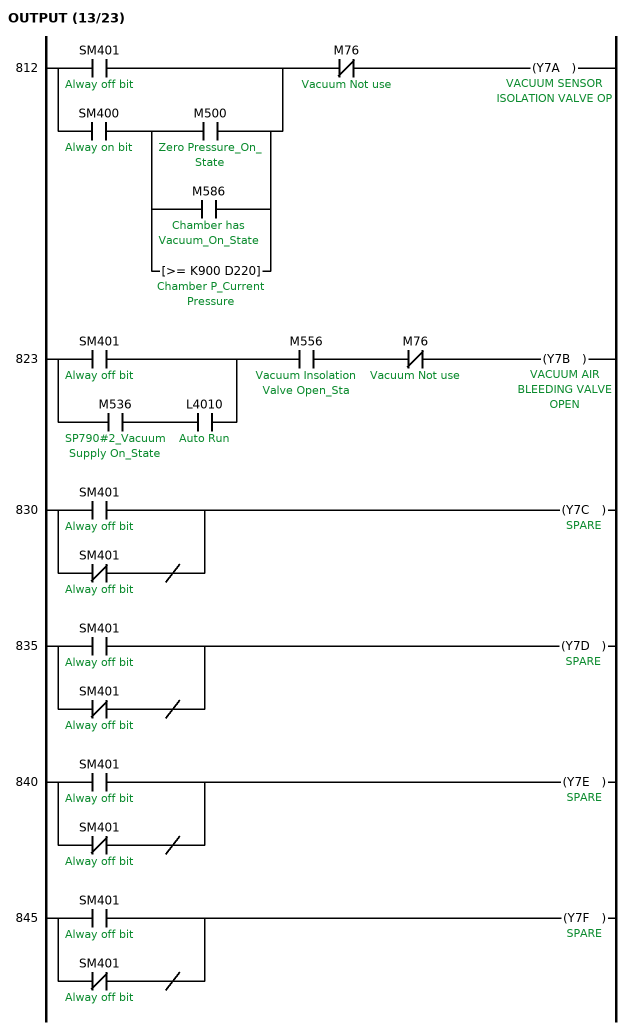
812   LD      SM401  ; Alway off bit
      LD      SM400  ; Alway on bit
      LD      M500  ; Zero Pressure_On_State
      OR      M586  ; Chamber has Vacuum_On_State
      OR>=    K900 D220  ; Chamber P_Current Pressure
      ANB
      ORB
      ANI     M76  ; Vacuum Not use
      OUT     Y7A  ; VACUUM SENSOR ISOLATION VALVE OP
823   LD      SM401  ; Alway off bit
      LD      M536  ; SP790#2_Vacuum Supply On_State
      AND     L4010  ; Auto Run
      ORB
      AND     M556  ; Vacuum Insolation Valve Open_Sta
      ANI     M76  ; Vacuum Not use
      OUT     Y7B  ; VACUUM AIR BLEEDING VALVE OPEN
830   LD      SM401  ; Alway off bit
      LDI     SM401  ; Alway off bit
      INV
      ORB
      OUT     Y7C  ; SPARE
835   LD      SM401  ; Alway off bit
      LDI     SM401  ; Alway off bit
      INV
      ORB
      OUT     Y7D  ; SPARE
840   LD      SM401  ; Alway off bit
      LDI     SM401  ; Alway off bit
      INV
      ORB
      OUT     Y7E  ; SPARE
845   LD      SM401  ; Alway off bit
      LDI     SM401  ; Alway off bit
      INV
      ORB
      OUT     Y7F  ; SPARE
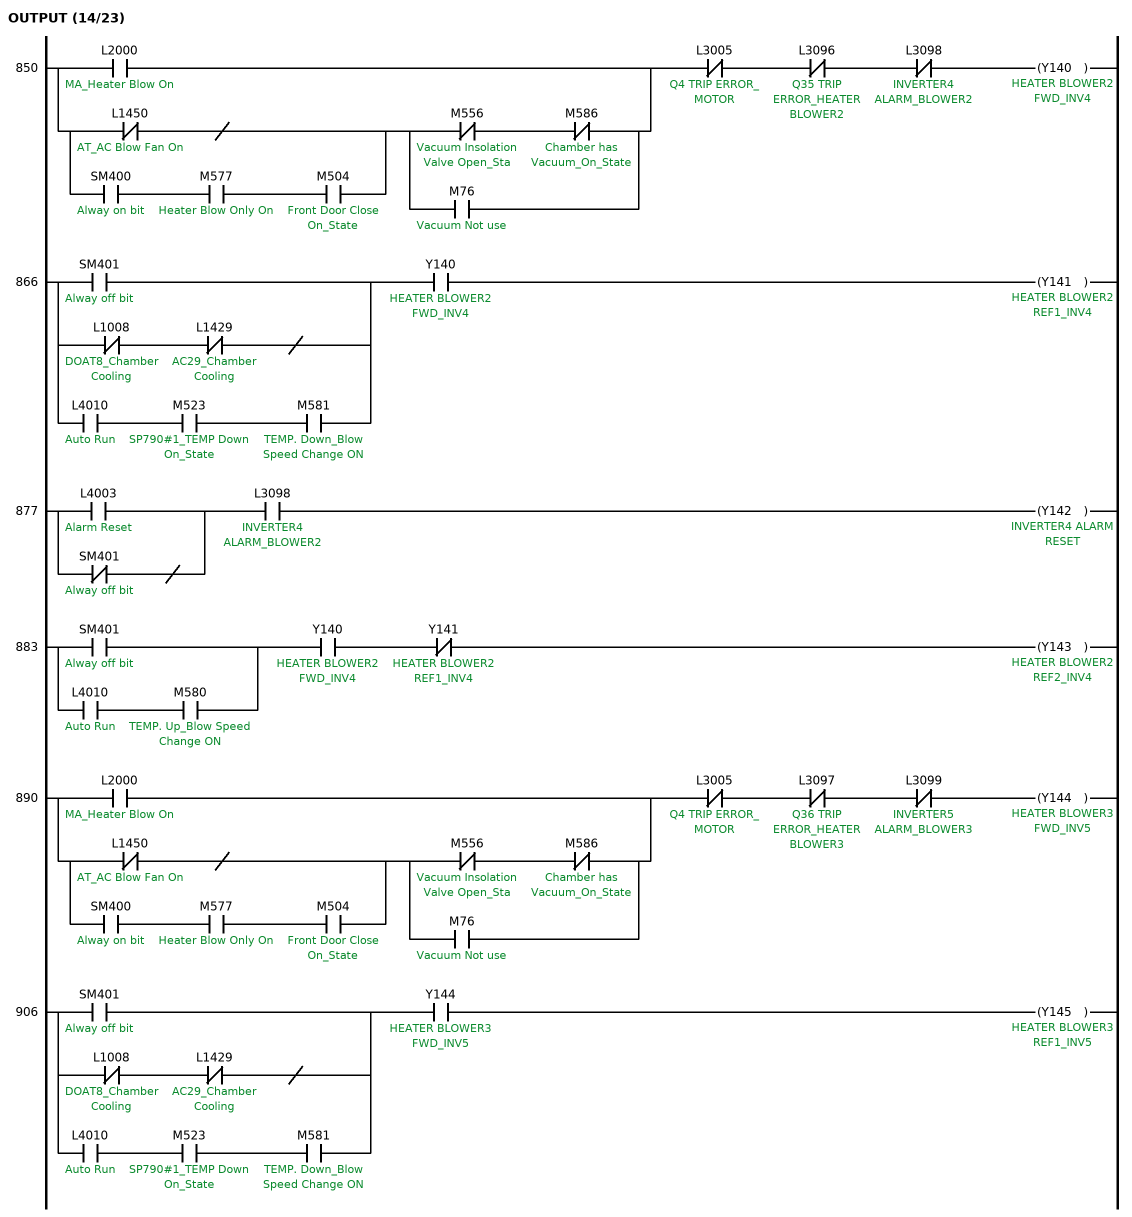
850   LD      L2000  ; MA_Heater Blow On
      LDI     L1450  ; AT_AC Blow Fan On
      INV
      LD      SM400  ; Alway on bit
      AND     M577  ; Heater Blow Only On
      AND     M504  ; Front Door Close On_State
      ORB
      LDI     M556  ; Vacuum Insolation Valve Open_Sta
      ANI     M586  ; Chamber has Vacuum_On_State
      OR      M76  ; Vacuum Not use
      ANB
      ORB
      ANI     L3005  ; Q4 TRIP ERROR_MOTOR
      ANI     L3096  ; Q35 TRIP ERROR_HEATER BLOWER2
      ANI     L3098  ; INVERTER4 ALARM_BLOWER2
      OUT     Y140  ; HEATER BLOWER2 FWD_INV4
866   LD      SM401  ; Alway off bit
      LDI     L1008  ; DOAT8_Chamber Cooling
      ANI     L1429  ; AC29_Chamber Cooling
      INV
      ORB
      LD      L4010  ; Auto Run
      AND     M523  ; SP790#1_TEMP Down On_State
      AND     M581  ; TEMP. Down_Blow Speed Change ON
      ORB
      AND     Y140  ; HEATER BLOWER2 FWD_INV4
      OUT     Y141  ; HEATER BLOWER2 REF1_INV4
877   LD      L4003  ; Alarm Reset
      LDI     SM401  ; Alway off bit
      INV
      ORB
      AND     L3098  ; INVERTER4 ALARM_BLOWER2
      OUT     Y142  ; INVERTER4 ALARM RESET
883   LD      SM401  ; Alway off bit
      LD      L4010  ; Auto Run
      AND     M580  ; TEMP. Up_Blow Speed Change ON
      ORB
      AND     Y140  ; HEATER BLOWER2 FWD_INV4
      ANI     Y141  ; HEATER BLOWER2 REF1_INV4
      OUT     Y143  ; HEATER BLOWER2 REF2_INV4
890   LD      L2000  ; MA_Heater Blow On
      LDI     L1450  ; AT_AC Blow Fan On
      INV
      LD      SM400  ; Alway on bit
      AND     M577  ; Heater Blow Only On
      AND     M504  ; Front Door Close On_State
      ORB
      LDI     M556  ; Vacuum Insolation Valve Open_Sta
      ANI     M586  ; Chamber has Vacuum_On_State
      OR      M76  ; Vacuum Not use
      ANB
      ORB
      ANI     L3005  ; Q4 TRIP ERROR_MOTOR
      ANI     L3097  ; Q36 TRIP ERROR_HEATER BLOWER3
      ANI     L3099  ; INVERTER5 ALARM_BLOWER3
      OUT     Y144  ; HEATER BLOWER3 FWD_INV5
906   LD      SM401  ; Alway off bit
      LDI     L1008  ; DOAT8_Chamber Cooling
      ANI     L1429  ; AC29_Chamber Cooling
      INV
      ORB
      LD      L4010  ; Auto Run
      AND     M523  ; SP790#1_TEMP Down On_State
      AND     M581  ; TEMP. Down_Blow Speed Change ON
      ORB
      AND     Y144  ; HEATER BLOWER3 FWD_INV5
      OUT     Y145  ; HEATER BLOWER3 REF1_INV5
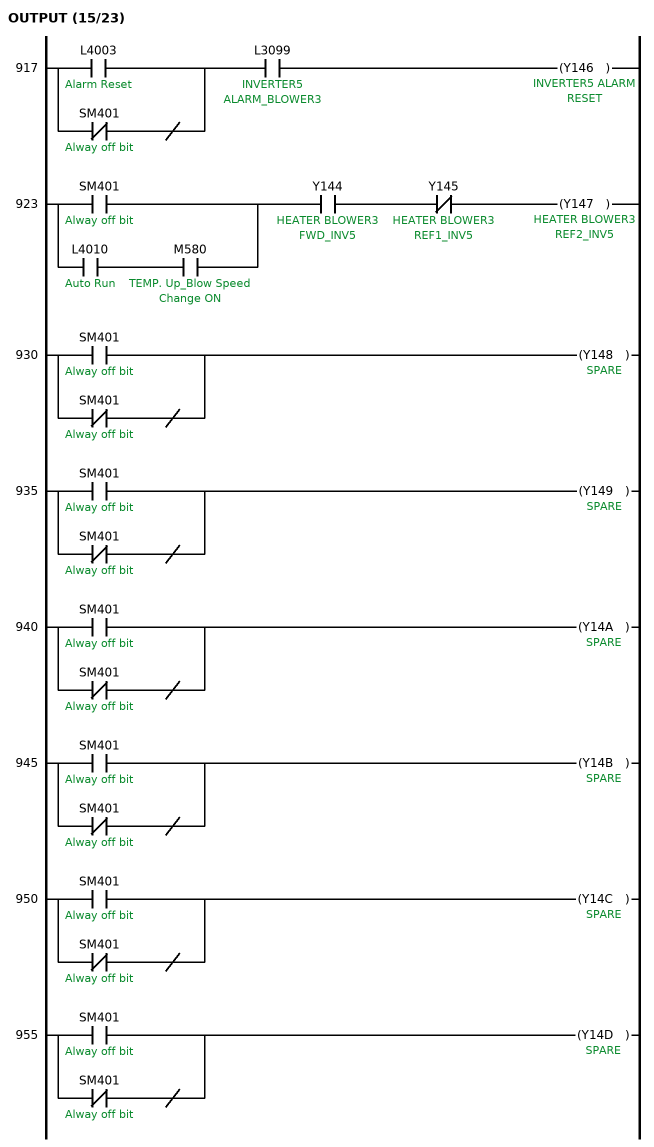
917   LD      L4003  ; Alarm Reset
      LDI     SM401  ; Alway off bit
      INV
      ORB
      AND     L3099  ; INVERTER5 ALARM_BLOWER3
      OUT     Y146  ; INVERTER5 ALARM RESET
923   LD      SM401  ; Alway off bit
      LD      L4010  ; Auto Run
      AND     M580  ; TEMP. Up_Blow Speed Change ON
      ORB
      AND     Y144  ; HEATER BLOWER3 FWD_INV5
      ANI     Y145  ; HEATER BLOWER3 REF1_INV5
      OUT     Y147  ; HEATER BLOWER3 REF2_INV5
930   LD      SM401  ; Alway off bit
      LDI     SM401  ; Alway off bit
      INV
      ORB
      OUT     Y148  ; SPARE
935   LD      SM401  ; Alway off bit
      LDI     SM401  ; Alway off bit
      INV
      ORB
      OUT     Y149  ; SPARE
940   LD      SM401  ; Alway off bit
      LDI     SM401  ; Alway off bit
      INV
      ORB
      OUT     Y14A  ; SPARE
945   LD      SM401  ; Alway off bit
      LDI     SM401  ; Alway off bit
      INV
      ORB
      OUT     Y14B  ; SPARE
950   LD      SM401  ; Alway off bit
      LDI     SM401  ; Alway off bit
      INV
      ORB
      OUT     Y14C  ; SPARE
955   LD      SM401  ; Alway off bit
      LDI     SM401  ; Alway off bit
      INV
      ORB
      OUT     Y14D  ; SPARE
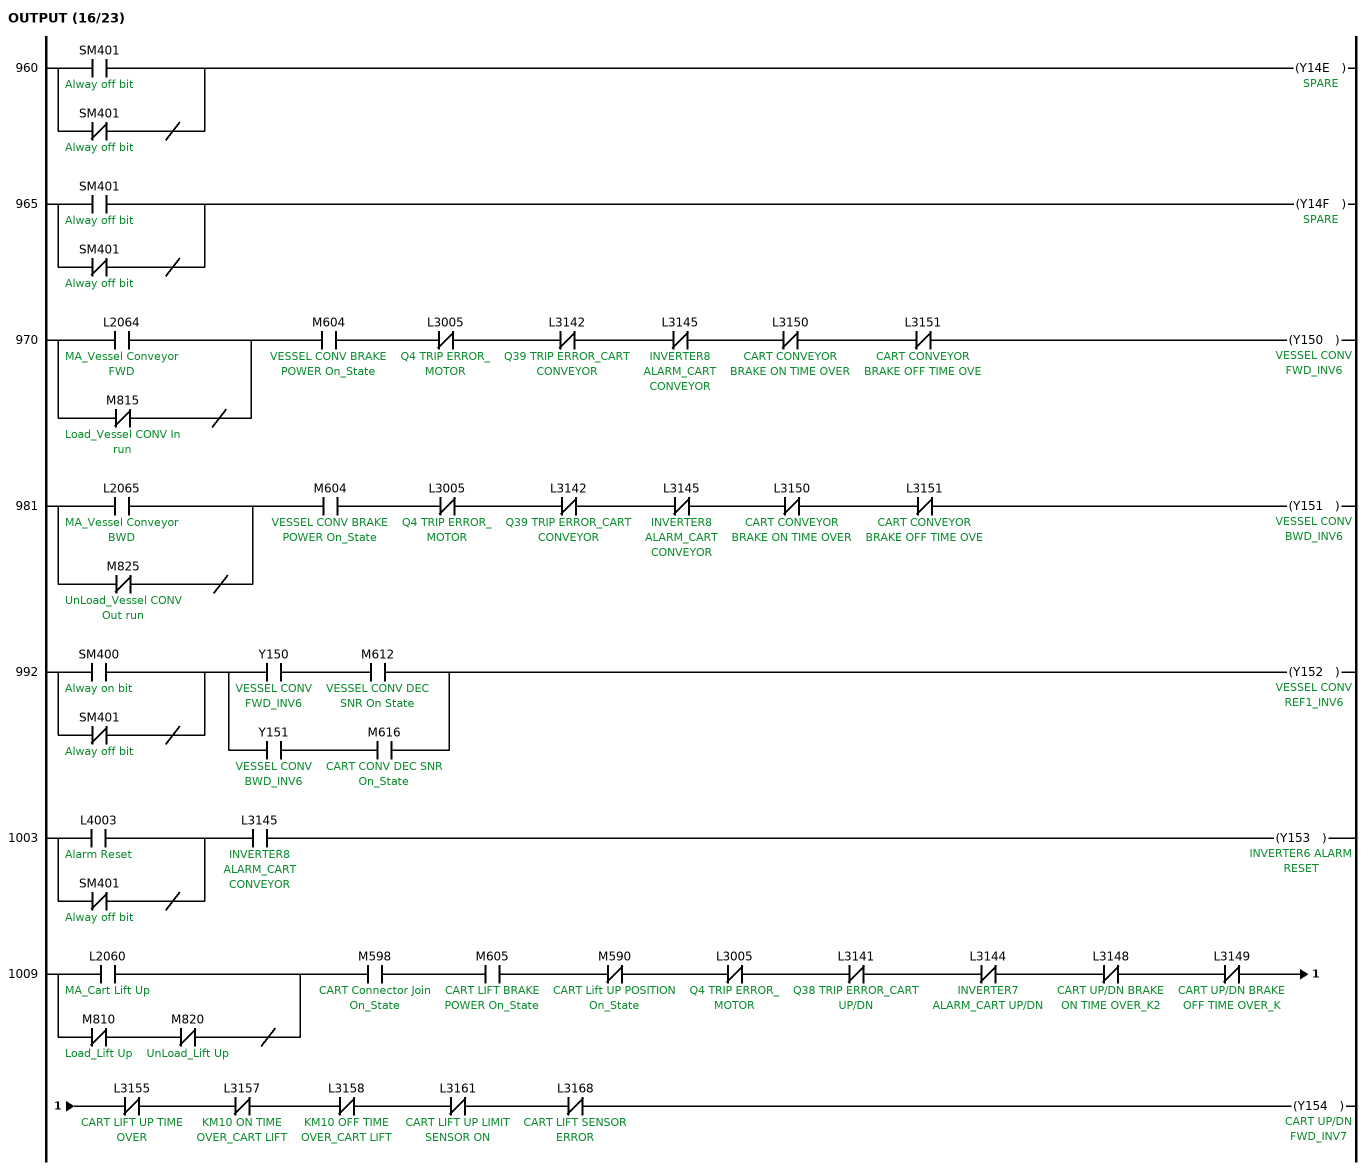
960   LD      SM401  ; Alway off bit
      LDI     SM401  ; Alway off bit
      INV
      ORB
      OUT     Y14E  ; SPARE
965   LD      SM401  ; Alway off bit
      LDI     SM401  ; Alway off bit
      INV
      ORB
      OUT     Y14F  ; SPARE
970   LD      L2064  ; MA_Vessel Conveyor FWD
      LDI     M815  ; Load_Vessel CONV In run
      INV
      ORB
      AND     M604  ; VESSEL CONV BRAKE POWER On_State
      ANI     L3005  ; Q4 TRIP ERROR_MOTOR
      ANI     L3142  ; Q39 TRIP ERROR_CART CONVEYOR
      ANI     L3145  ; INVERTER8 ALARM_CART CONVEYOR
      ANI     L3150  ; CART CONVEYOR BRAKE ON TIME OVER
      ANI     L3151  ; CART CONVEYOR BRAKE OFF TIME OVE
      OUT     Y150  ; VESSEL CONV FWD_INV6
981   LD      L2065  ; MA_Vessel Conveyor BWD
      LDI     M825  ; UnLoad_Vessel CONV Out run
      INV
      ORB
      AND     M604  ; VESSEL CONV BRAKE POWER On_State
      ANI     L3005  ; Q4 TRIP ERROR_MOTOR
      ANI     L3142  ; Q39 TRIP ERROR_CART CONVEYOR
      ANI     L3145  ; INVERTER8 ALARM_CART CONVEYOR
      ANI     L3150  ; CART CONVEYOR BRAKE ON TIME OVER
      ANI     L3151  ; CART CONVEYOR BRAKE OFF TIME OVE
      OUT     Y151  ; VESSEL CONV BWD_INV6
992   LD      SM400  ; Alway on bit
      LDI     SM401  ; Alway off bit
      INV
      ORB
      LD      Y150  ; VESSEL CONV FWD_INV6
      AND     M612  ; VESSEL CONV DEC SNR On State
      LD      Y151  ; VESSEL CONV BWD_INV6
      AND     M616  ; CART CONV DEC SNR On_State
      ORB
      ANB
      OUT     Y152  ; VESSEL CONV REF1_INV6
1003  LD      L4003  ; Alarm Reset
      LDI     SM401  ; Alway off bit
      INV
      ORB
      AND     L3145  ; INVERTER8 ALARM_CART CONVEYOR
      OUT     Y153  ; INVERTER6 ALARM RESET
1009  LD      L2060  ; MA_Cart Lift Up
      LDI     M810  ; Load_Lift Up
      ANI     M820  ; UnLoad_Lift Up
      INV
      ORB
      AND     M598  ; CART Connector Join On_State
      AND     M605  ; CART LIFT BRAKE POWER On_State
      ANI     M590  ; CART Lift UP POSITION On_State
      ANI     L3005  ; Q4 TRIP ERROR_MOTOR
      ANI     L3141  ; Q38 TRIP ERROR_CART UP/DN
      ANI     L3144  ; INVERTER7 ALARM_CART UP/DN
      ANI     L3148  ; CART UP/DN BRAKE ON TIME OVER_K2
      ANI     L3149  ; CART UP/DN BRAKE OFF TIME OVER_K
      ANI     L3155  ; CART LIFT UP TIME OVER
      ANI     L3157  ; KM10 ON TIME OVER_CART LIFT
      ANI     L3158  ; KM10 OFF TIME OVER_CART LIFT
      ANI     L3161  ; CART LIFT UP LIMIT SENSOR ON
      ANI     L3168  ; CART LIFT SENSOR ERROR
      OUT     Y154  ; CART UP/DN FWD_INV7
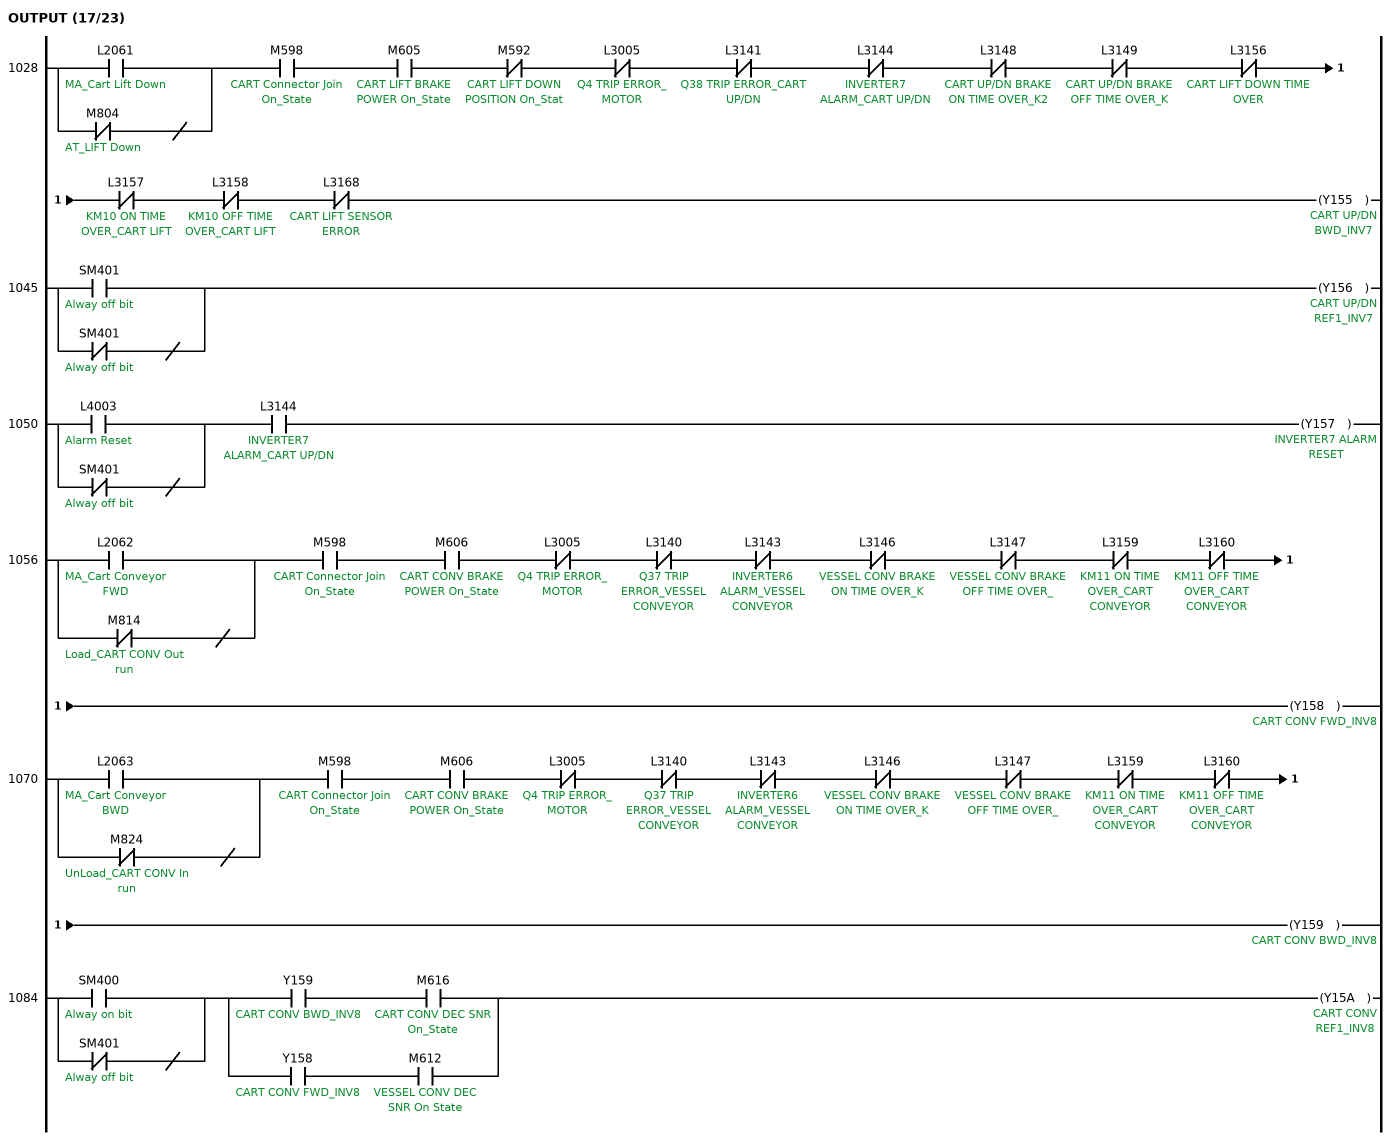
1028  LD      L2061  ; MA_Cart Lift Down
      LDI     M804  ; AT_LIFT Down
      INV
      ORB
      AND     M598  ; CART Connector Join On_State
      AND     M605  ; CART LIFT BRAKE POWER On_State
      ANI     M592  ; CART LIFT DOWN  POSITION On_Stat
      ANI     L3005  ; Q4 TRIP ERROR_MOTOR
      ANI     L3141  ; Q38 TRIP ERROR_CART UP/DN
      ANI     L3144  ; INVERTER7 ALARM_CART UP/DN
      ANI     L3148  ; CART UP/DN BRAKE ON TIME OVER_K2
      ANI     L3149  ; CART UP/DN BRAKE OFF TIME OVER_K
      ANI     L3156  ; CART LIFT DOWN TIME OVER
      ANI     L3157  ; KM10 ON TIME OVER_CART LIFT
      ANI     L3158  ; KM10 OFF TIME OVER_CART LIFT
      ANI     L3168  ; CART LIFT SENSOR ERROR
      OUT     Y155  ; CART UP/DN BWD_INV7
1045  LD      SM401  ; Alway off bit
      LDI     SM401  ; Alway off bit
      INV
      ORB
      OUT     Y156  ; CART UP/DN REF1_INV7
1050  LD      L4003  ; Alarm Reset
      LDI     SM401  ; Alway off bit
      INV
      ORB
      AND     L3144  ; INVERTER7 ALARM_CART UP/DN
      OUT     Y157  ; INVERTER7 ALARM RESET
1056  LD      L2062  ; MA_Cart Conveyor FWD
      LDI     M814  ; Load_CART CONV Out run
      INV
      ORB
      AND     M598  ; CART Connector Join On_State
      AND     M606  ; CART CONV BRAKE POWER On_State
      ANI     L3005  ; Q4 TRIP ERROR_MOTOR
      ANI     L3140  ; Q37 TRIP ERROR_VESSEL CONVEYOR
      ANI     L3143  ; INVERTER6 ALARM_VESSEL CONVEYOR
      ANI     L3146  ; VESSEL CONV BRAKE ON TIME OVER_K
      ANI     L3147  ; VESSEL CONV BRAKE OFF TIME OVER_
      ANI     L3159  ; KM11 ON TIME OVER_CART CONVEYOR
      ANI     L3160  ; KM11 OFF TIME OVER_CART CONVEYOR
      OUT     Y158  ; CART CONV FWD_INV8
1070  LD      L2063  ; MA_Cart Conveyor BWD
      LDI     M824  ; UnLoad_CART CONV In run
      INV
      ORB
      AND     M598  ; CART Connector Join On_State
      AND     M606  ; CART CONV BRAKE POWER On_State
      ANI     L3005  ; Q4 TRIP ERROR_MOTOR
      ANI     L3140  ; Q37 TRIP ERROR_VESSEL CONVEYOR
      ANI     L3143  ; INVERTER6 ALARM_VESSEL CONVEYOR
      ANI     L3146  ; VESSEL CONV BRAKE ON TIME OVER_K
      ANI     L3147  ; VESSEL CONV BRAKE OFF TIME OVER_
      ANI     L3159  ; KM11 ON TIME OVER_CART CONVEYOR
      ANI     L3160  ; KM11 OFF TIME OVER_CART CONVEYOR
      OUT     Y159  ; CART CONV BWD_INV8
1084  LD      SM400  ; Alway on bit
      LDI     SM401  ; Alway off bit
      INV
      ORB
      LD      Y159  ; CART CONV BWD_INV8
      AND     M616  ; CART CONV DEC SNR On_State
      LD      Y158  ; CART CONV FWD_INV8
      AND     M612  ; VESSEL CONV DEC SNR On State
      ORB
      ANB
      OUT     Y15A  ; CART CONV REF1_INV8
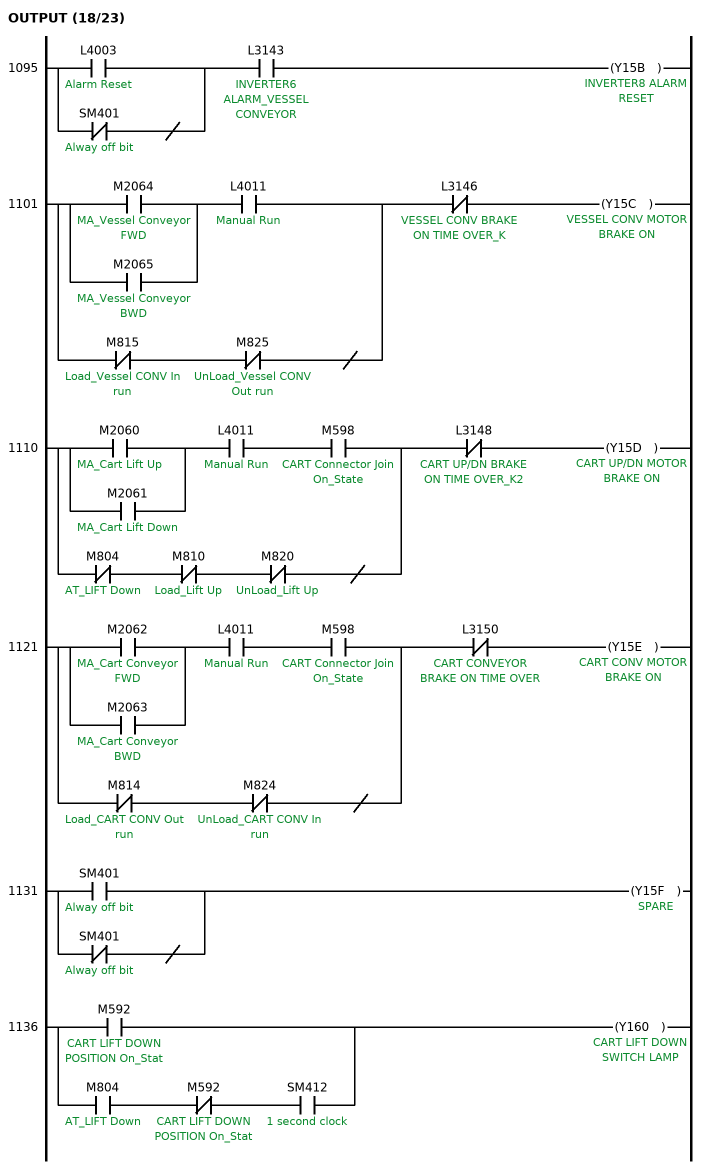
1095  LD      L4003  ; Alarm Reset
      LDI     SM401  ; Alway off bit
      INV
      ORB
      AND     L3143  ; INVERTER6 ALARM_VESSEL CONVEYOR
      OUT     Y15B  ; INVERTER8 ALARM RESET
1101  LD      M2064  ; MA_Vessel Conveyor FWD
      OR      M2065  ; MA_Vessel Conveyor BWD
      AND     L4011  ; Manual Run
      LDI     M815  ; Load_Vessel CONV In run
      ANI     M825  ; UnLoad_Vessel CONV Out run
      INV
      ORB
      ANI     L3146  ; VESSEL CONV BRAKE ON TIME OVER_K
      OUT     Y15C  ; VESSEL CONV MOTOR BRAKE ON
1110  LD      M2060  ; MA_Cart Lift Up
      OR      M2061  ; MA_Cart Lift Down
      AND     L4011  ; Manual Run
      AND     M598  ; CART Connector Join On_State
      LDI     M804  ; AT_LIFT Down
      ANI     M810  ; Load_Lift Up
      ANI     M820  ; UnLoad_Lift Up
      INV
      ORB
      ANI     L3148  ; CART UP/DN BRAKE ON TIME OVER_K2
      OUT     Y15D  ; CART UP/DN MOTOR BRAKE ON
1121  LD      M2062  ; MA_Cart Conveyor FWD
      OR      M2063  ; MA_Cart Conveyor BWD
      AND     L4011  ; Manual Run
      AND     M598  ; CART Connector Join On_State
      LDI     M814  ; Load_CART CONV Out run
      ANI     M824  ; UnLoad_CART CONV In run
      INV
      ORB
      ANI     L3150  ; CART CONVEYOR BRAKE ON TIME OVER
      OUT     Y15E  ; CART CONV MOTOR BRAKE ON
1131  LD      SM401  ; Alway off bit
      LDI     SM401  ; Alway off bit
      INV
      ORB
      OUT     Y15F  ; SPARE
1136  LD      M592  ; CART LIFT DOWN  POSITION On_Stat
      LD      M804  ; AT_LIFT Down
      ANI     M592  ; CART LIFT DOWN  POSITION On_Stat
      AND     SM412  ; 1 second clock
      ORB
      OUT     Y160  ; CART LIFT DOWN SWITCH LAMP
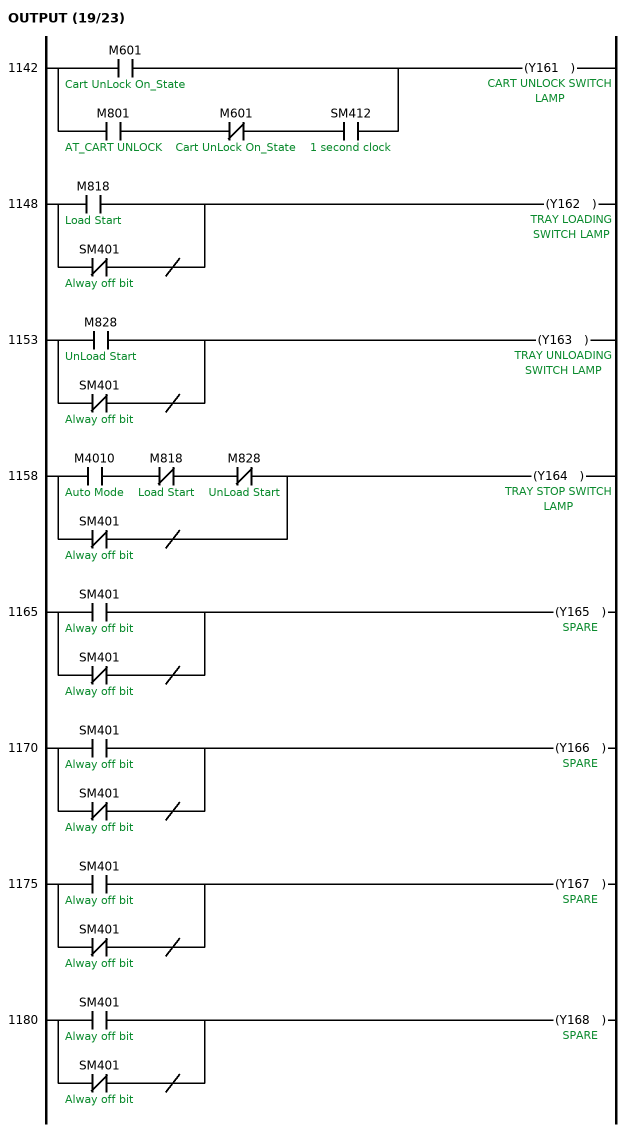
1142  LD      M601  ; Cart UnLock On_State
      LD      M801  ; AT_CART UNLOCK
      ANI     M601  ; Cart UnLock On_State
      AND     SM412  ; 1 second clock
      ORB
      OUT     Y161  ; CART UNLOCK SWITCH LAMP
1148  LD      M818  ; Load Start
      LDI     SM401  ; Alway off bit
      INV
      ORB
      OUT     Y162  ; TRAY LOADING SWITCH LAMP
1153  LD      M828  ; UnLoad Start
      LDI     SM401  ; Alway off bit
      INV
      ORB
      OUT     Y163  ; TRAY UNLOADING SWITCH LAMP
1158  LD      M4010  ; Auto Mode
      ANI     M818  ; Load Start
      ANI     M828  ; UnLoad Start
      LDI     SM401  ; Alway off bit
      INV
      ORB
      OUT     Y164  ; TRAY STOP SWITCH LAMP
1165  LD      SM401  ; Alway off bit
      LDI     SM401  ; Alway off bit
      INV
      ORB
      OUT     Y165  ; SPARE
1170  LD      SM401  ; Alway off bit
      LDI     SM401  ; Alway off bit
      INV
      ORB
      OUT     Y166  ; SPARE
1175  LD      SM401  ; Alway off bit
      LDI     SM401  ; Alway off bit
      INV
      ORB
      OUT     Y167  ; SPARE
1180  LD      SM401  ; Alway off bit
      LDI     SM401  ; Alway off bit
      INV
      ORB
      OUT     Y168  ; SPARE
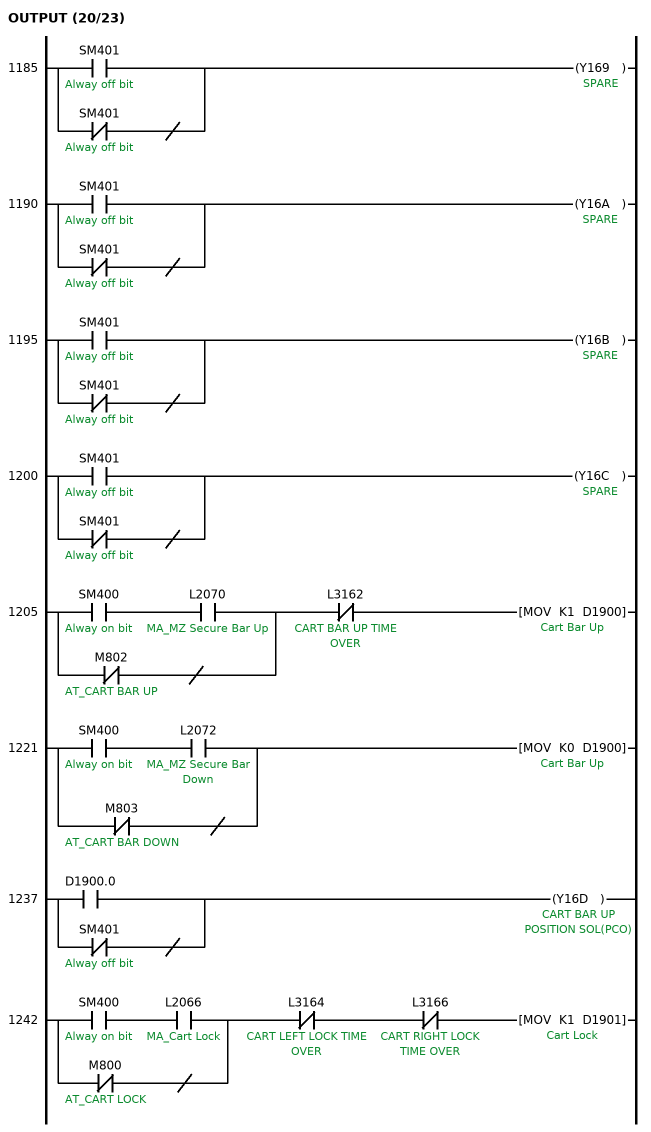
1185  LD      SM401  ; Alway off bit
      LDI     SM401  ; Alway off bit
      INV
      ORB
      OUT     Y169  ; SPARE
1190  LD      SM401  ; Alway off bit
      LDI     SM401  ; Alway off bit
      INV
      ORB
      OUT     Y16A  ; SPARE
1195  LD      SM401  ; Alway off bit
      LDI     SM401  ; Alway off bit
      INV
      ORB
      OUT     Y16B  ; SPARE
1200  LD      SM401  ; Alway off bit
      LDI     SM401  ; Alway off bit
      INV
      ORB
      OUT     Y16C  ; SPARE
1205  LD      SM400  ; Alway on bit
      AND     L2070  ; MA_MZ Secure Bar Up
      LDI     M802  ; AT_CART BAR UP
      INV
      ORB
      ANI     L3162  ; CART BAR UP TIME OVER
      MOV     K1 D1900  ; Cart Bar Up
        [note] Cart Bar Up
1221  LD      SM400  ; Alway on bit
      AND     L2072  ; MA_MZ Secure Bar Down
      LDI     M803  ; AT_CART BAR DOWN
      INV
      ORB
      MOV     K0 D1900
        [note] Cart Bar Down
1237  LD      D1900.0
      LDI     SM401  ; Alway off bit
      INV
      ORB
      OUT     Y16D  ; CART BAR UP POSITION SOL(PCO)
1242  LD      SM400  ; Alway on bit
      AND     L2066  ; MA_Cart Lock
      LDI     M800  ; AT_CART LOCK
      INV
      ORB
      ANI     L3164  ; CART LEFT LOCK TIME OVER
      ANI     L3166  ; CART RIGHT LOCK TIME OVER
      MOV     K1 D1901  ; Cart Lock
        [note] Cart Lock
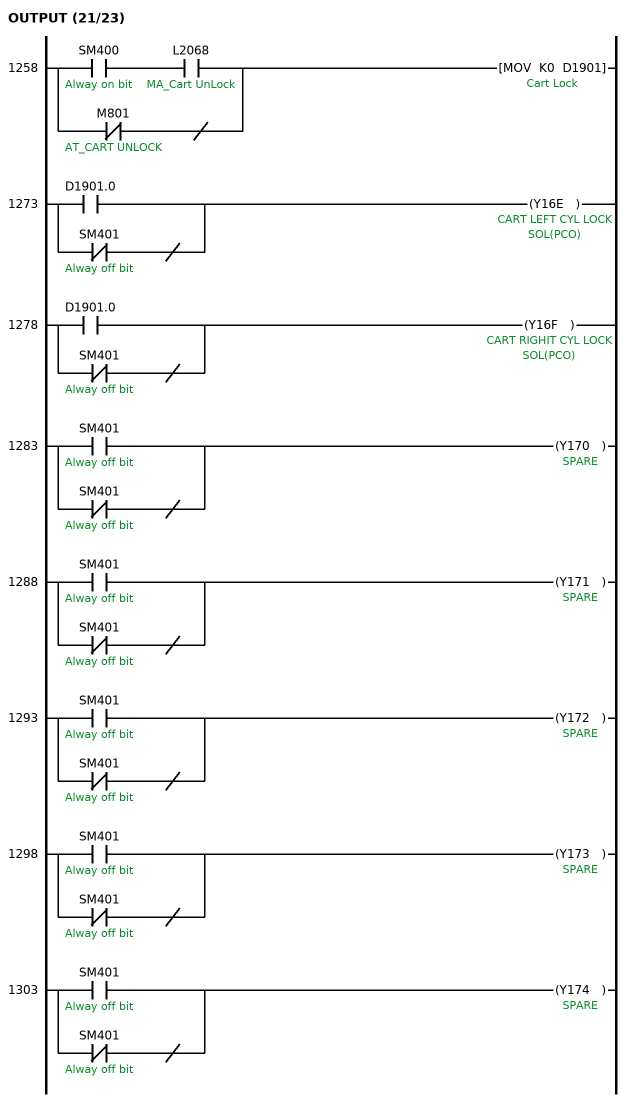
1258  LD      SM400  ; Alway on bit
      AND     L2068  ; MA_Cart UnLock
      LDI     M801  ; AT_CART UNLOCK
      INV
      ORB
      MOV     K0 D1901
        [note] Cart Unlock
1273  LD      D1901.0
      LDI     SM401  ; Alway off bit
      INV
      ORB
      OUT     Y16E  ; CART LEFT CYL LOCK SOL(PCO)
1278  LD      D1901.0
      LDI     SM401  ; Alway off bit
      INV
      ORB
      OUT     Y16F  ; CART RIGHIT CYL LOCK SOL(PCO)
1283  LD      SM401  ; Alway off bit
      LDI     SM401  ; Alway off bit
      INV
      ORB
      OUT     Y170  ; SPARE
1288  LD      SM401  ; Alway off bit
      LDI     SM401  ; Alway off bit
      INV
      ORB
      OUT     Y171  ; SPARE
1293  LD      SM401  ; Alway off bit
      LDI     SM401  ; Alway off bit
      INV
      ORB
      OUT     Y172  ; SPARE
1298  LD      SM401  ; Alway off bit
      LDI     SM401  ; Alway off bit
      INV
      ORB
      OUT     Y173  ; SPARE
1303  LD      SM401  ; Alway off bit
      LDI     SM401  ; Alway off bit
      INV
      ORB
      OUT     Y174  ; SPARE
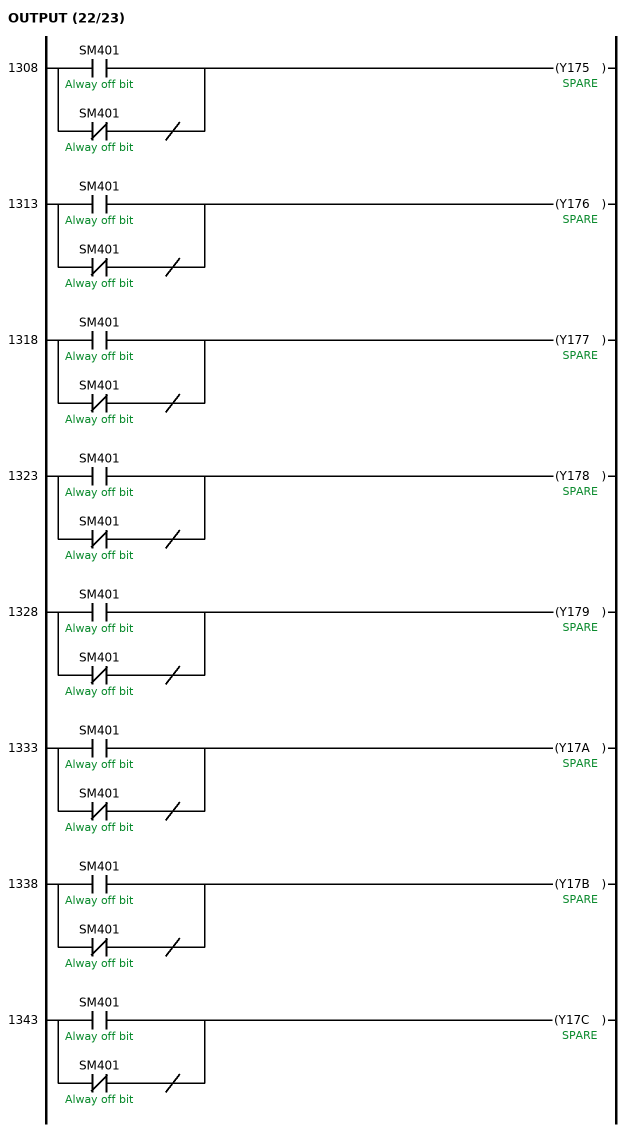
1308  LD      SM401  ; Alway off bit
      LDI     SM401  ; Alway off bit
      INV
      ORB
      OUT     Y175  ; SPARE
1313  LD      SM401  ; Alway off bit
      LDI     SM401  ; Alway off bit
      INV
      ORB
      OUT     Y176  ; SPARE
1318  LD      SM401  ; Alway off bit
      LDI     SM401  ; Alway off bit
      INV
      ORB
      OUT     Y177  ; SPARE
1323  LD      SM401  ; Alway off bit
      LDI     SM401  ; Alway off bit
      INV
      ORB
      OUT     Y178  ; SPARE
1328  LD      SM401  ; Alway off bit
      LDI     SM401  ; Alway off bit
      INV
      ORB
      OUT     Y179  ; SPARE
1333  LD      SM401  ; Alway off bit
      LDI     SM401  ; Alway off bit
      INV
      ORB
      OUT     Y17A  ; SPARE
1338  LD      SM401  ; Alway off bit
      LDI     SM401  ; Alway off bit
      INV
      ORB
      OUT     Y17B  ; SPARE
1343  LD      SM401  ; Alway off bit
      LDI     SM401  ; Alway off bit
      INV
      ORB
      OUT     Y17C  ; SPARE
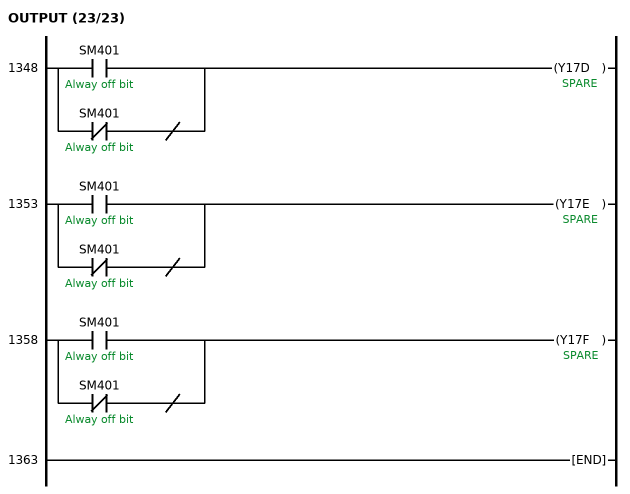
1348  LD      SM401  ; Alway off bit
      LDI     SM401  ; Alway off bit
      INV
      ORB
      OUT     Y17D  ; SPARE
1353  LD      SM401  ; Alway off bit
      LDI     SM401  ; Alway off bit
      INV
      ORB
      OUT     Y17E  ; SPARE
1358  LD      SM401  ; Alway off bit
      LDI     SM401  ; Alway off bit
      INV
      ORB
      OUT     Y17F  ; SPARE
1363  END
END_PROGRAM
